	IF arrBetrartHandAktiv[I_nSchutzBer]
		THEN
			stUniAnstgFkt.arrGrdstFkt[0]:= I_arrZuwGrdstFkt[0];
			stUniAnstgFkt.arrGrdstFkt[1]:= I_arrZuwGrdstFkt[1];
			stUniAnstgFkt.arrGrdstFkt[2]:= I_arrZuwGrdstFkt[2];
			stUniAnstgFkt.arrGrdstFkt[3]:= I_arrZuwGrdstFkt[3];
		ELSE
			stUniAnstgFkt.arrGrdstFkt[0]:= 
			stUniAnstgFkt.arrGrdstFkt[1]:=
			stUniAnstgFkt.arrGrdstFkt[2]:=
			stUniAnstgFkt.arrGrdstFkt[3]:= FALSE;
   END_IF
	IF arrBetrartAutomAktiv[I_nSchutzBer] OR TRUE //ToDo
		THEN
			stUniAnstgFkt.arrAutomFkt[0]:= I_arrZuwAutomFkt[0];
			stUniAnstgFkt.arrAutomFkt[1]:= I_arrZuwAutomFkt[1];
			stUniAnstgFkt.arrAutomFkt[2]:= I_arrZuwAutomFkt[2];
			stUniAnstgFkt.arrAutomFkt[3]:= I_arrZuwAutomFkt[3];
		ELSE
			stUniAnstgFkt.arrAutomFkt[0]:= 
			stUniAnstgFkt.arrAutomFkt[1]:= 
			stUniAnstgFkt.arrAutomFkt[2]:= 
			stUniAnstgFkt.arrAutomFkt[3]:= FALSE;
   END_IF

	(**************************************************)	

	stUniAnstgFkt.arrFktAusfg[0]:= stUniAnstgFkt.arrGrdstFkt[0]
										 	 OR stUniAnstgFkt.arrHandFkt[0]
										 	 OR stUniAnstgFkt.arrAutomFkt[0];

	stUniAnstgFkt.arrFktAusfg[1]:= stUniAnstgFkt.arrGrdstFkt[1]
										 	 OR stUniAnstgFkt.arrHandFkt[1]
										 	 OR stUniAnstgFkt.arrAutomFkt[1];

	stUniAnstgFkt.arrFktAusfg[2]:= stUniAnstgFkt.arrGrdstFkt[2]
										 	 OR stUniAnstgFkt.arrHandFkt[2]
										 	 OR stUniAnstgFkt.arrAutomFkt[2];

	stUniAnstgFkt.arrFktAusfg[3]:= stUniAnstgFkt.arrGrdstFkt[3]
										 	 OR stUniAnstgFkt.arrHandFkt[3]
										 	 OR stUniAnstgFkt.arrAutomFkt[3];

	(**************************************************)
END_ACTION

ACTION c_Verstellg:
	(*Antriebstyp "Verstellg." /z.B. FU-Antriebe mit Eil/Schleichbewegung...*)

	(*Verwendete Softkeytasten = 5 (s.Beispiel)*)

   (*       "Handfunktion"       /   "Softkeytaste 1"   /   "Softkeytaste 2"   /   "Softkeytaste 3"   /   "Softkeytaste 4"   /   "Softkeytaste 5"   *)
	(*                                                                          															  								 *) 
	(*----- Verstellantrieb ------/_____zurückfahren_____/_______vorfahren______/_______langsam________/_______schnell________/________Reset_________*)

	(*Softkeyleiste.1		:Funktion ein.-ausschalten Reversierend*)
	(*Softkeyleiste.2		:Funktion ein.-ausschalten             *)
	(*Softkeyleiste.3		:Funktion langsame Drehzahl (SollwMin) *)
	(*Softkeyleiste.4		:Funktion schnelle Drehzahl (SollwVrg) *)
	(*Softkeyleiste.5		:Platzhalter									 *)

	(*Hinweis:
	- Funktion wird durch "VerrHdFkt" gesperrt (z.B. bei Überstandserkennung...)
	- Funktion wird durch "EndlHdFkt/VerzHdFkt" zurückgenommen bzw. umgeschaltet
	*)
	
	(**************************************************)	

	stUniAnstgFkt.bHandAnw0:= IQ_stUniAnstgHMI.stHandFktHMI[1].bySwitch > 0;
	stUniAnstgFkt.bHandAnw1:= IQ_stUniAnstgHMI.stHandFktHMI[2].bySwitch > 0;
	stUniAnstgFkt.bHandAnw2:= IQ_stUniAnstgHMI.stHandFktHMI[3].bySwitch > 0;
	stUniAnstgFkt.bHandAnw3:= IQ_stUniAnstgHMI.stHandFktHMI[4].bySwitch > 0;
	
	IF arrBetrartAutomAktiv[I_nSchutzBer]
		OR I_bResHandFkt
		OR NOT I_bExtReglFrg
		THEN
			stUniAnstgFkt.arrHandFkt[0]:=
			stUniAnstgFkt.arrHandFkt[1]:=
			stUniAnstgFkt.arrHandFkt[2]:=
			stUniAnstgFkt.arrHandFkt[3]:= FALSE;
		ELSE
			IF NOT arrBetrartAutomSpeichn[I_nSchutzBer]
				THEN
					IF NOT arrGrdstlgBetrAktiv[I_nSchutzBer]
						THEN
							 rtrigHandFkt1 (CLK:= stUniAnstgFkt.bHandAnw1);
							 IF rtrigHandFkt1.Q THEN
								 stUniAnstgFkt.arrHandFkt[1]:= NOT stUniAnstgFkt.arrHandFkt[1];
							 END_IF
							 IF NOT arrBetrartHandAktiv[I_nSchutzBer]
								 OR stUniAnstgFkt.arrHandFkt[0]
								 OR I_bVerrHdFktV OR NOT I_bEndlHdFktV THEN
								 stUniAnstgFkt.arrHandFkt[1]:= FALSE;
							 END_IF
	 
							 rtrigHandFkt0 (CLK:= stUniAnstgFkt.bHandAnw0);
							 IF rtrigHandFkt0.Q THEN
								 stUniAnstgFkt.arrHandFkt[0]:= NOT stUniAnstgFkt.arrHandFkt[0];
							 END_IF
							 IF NOT arrBetrartHandAktiv[I_nSchutzBer]
								 OR stUniAnstgFkt.arrHandFkt[1]
								 OR I_bVerrHdFktZ OR NOT I_bEndlHdFktZ THEN
								 stUniAnstgFkt.arrHandFkt[0]:= FALSE;
							 END_IF
	 
							 IF stUniAnstgFkt.bHandAnw3 THEN
								 stUniAnstgFkt.arrHandFkt[3]:= TRUE;
							 END_IF
							 IF NOT arrBetrartHandAktiv[I_nSchutzBer]
								 OR (stUniAnstgFkt.arrHandFkt[1] AND I_bVerzHdFktV)
								 OR (stUniAnstgFkt.arrHandFkt[0] AND I_bVerzHdFktZ)
								 OR stUniAnstgFkt.bHandAnw2 THEN
								 stUniAnstgFkt.arrHandFkt[3]:= FALSE;
							 END_IF
					END_IF
			END_IF
	END_IF

	IF arrBetrartHandAktiv[I_nSchutzBer]
		THEN
			stUniAnstgFkt.nHandStat:= 0;			(*Funktion freigegeben*)
			IF stUniAnstgFkt.arrHandFkt[1]
				THEN
					stUniAnstgFkt.nHandStat:= 2;	(*Handfunktion.2 aktiv*)
			END_IF
			IF stUniAnstgFkt.arrHandFkt[0]
				THEN
					stUniAnstgFkt.nHandStat:= 1;	(*Handfunktion.1 aktiv*)
			END_IF
			IF stUniAnstgFkt.arrHandFkt[3]
				THEN
					stUniAnstgFkt.nHandStat:=
					stUniAnstgFkt.nHandStat + 8;	(*Handfunktion.4 aktiv*)
				ELSE
					stUniAnstgFkt.nHandStat:=
					stUniAnstgFkt.nHandStat + 4;	(*Handfunktion.3 aktiv*)
			END_IF
		ELSE
			stUniAnstgFkt.nHandStat:= 256;		(*Funktion gesperrt*)
	END_IF

	(**************************************************)	

	IF arrBetrartHandAktiv[I_nSchutzBer]
		THEN
			stUniAnstgFkt.arrGrdstFkt[0]:= I_arrZuwGrdstFkt[0];
			stUniAnstgFkt.arrGrdstFkt[1]:= I_arrZuwGrdstFkt[1];
			stUniAnstgFkt.arrGrdstFkt[3]:= I_arrZuwGrdstFkt[2];
		ELSE
			stUniAnstgFkt.arrGrdstFkt[0]:= 
			stUniAnstgFkt.arrGrdstFkt[1]:=
			stUniAnstgFkt.arrGrdstFkt[3]:= FALSE;
   END_IF
	IF arrBetrartAutomAktiv[I_nSchutzBer] OR TRUE //ToDo
		THEN
			stUniAnstgFkt.arrAutomFkt[0]:= I_arrZuwAutomFkt[0];
			stUniAnstgFkt.arrAutomFkt[1]:= I_arrZuwAutomFkt[1];
			stUniAnstgFkt.arrAutomFkt[3]:= I_arrZuwAutomFkt[2];
		ELSE
			stUniAnstgFkt.arrAutomFkt[0]:= 
			stUniAnstgFkt.arrAutomFkt[1]:= 
			stUniAnstgFkt.arrAutomFkt[3]:= FALSE;
   END_IF

	(**************************************************)	

	stUniAnstgFkt.arrFktAusfg[0]:= (stUniAnstgFkt.arrGrdstFkt[0]
										 	 	OR stUniAnstgFkt.arrHandFkt[0]
										 	 	OR stUniAnstgFkt.arrAutomFkt[0])
											AND I_bEndlHdFktZ;

	stUniAnstgFkt.arrFktAusfg[1]:= (stUniAnstgFkt.arrGrdstFkt[1]
										 	 OR stUniAnstgFkt.arrHandFkt[1]
										 	 OR stUniAnstgFkt.arrAutomFkt[1])
											AND I_bEndlHdFktV;

	stUniAnstgFkt.arrFktAusfg[3]:= (stUniAnstgFkt.arrGrdstFkt[3]
												 OR stUniAnstgFkt.arrHandFkt[3]
												 OR stUniAnstgFkt.arrAutomFkt[3])
											AND(( stUniAnstgFkt.arrFktAusfg[0]
													AND NOT I_bVerzHdFktZ)
												OR ( stUniAnstgFkt.arrFktAusfg[1]
													AND NOT I_bVerzHdFktV));

	(**************************************************)
END_ACTION

ACTION d_EilSchleich:
	(*Antriebstyp "EilSchleich" /z.B. FU-Antriebe mit Eil/Schleichachse...*)

	(*Verwendete Softkeytasten = 5 (s.Beispiel)*)

   (*       "Handfunktion"       /   "Softkeytaste 1"   /   "Softkeytaste 2"   /   "Softkeytaste 3"   /   "Softkeytaste 4"   /   "Softkeytaste 5"   *)
	(*                                                                          															  								 *) 
	(*------ Verstellachse -------/____negativ fahren____/____positiv fahren____/_________Frei_________/_________Frei_________/________Reset_________*)
	
	(*Softkeyleiste.1		:Funktion Tastend aktiv /Richtg. Negativ*)
	(*Softkeyleiste.2		:Funktion Tastend aktiv /Richtg. Positiv*)
	(*Softkeyleiste.3		:Platzhalter				 					 *)
	(*Softkeyleiste.4		:Platzhalter				 					 *)
	(*Softkeyleiste.5		:Platzhalter									 *)

	(*Hinweis:
	- Funktion wird durch "VerrHdFkt" gesperrt (z.B. bei Überstandserkennung...)
	*)

	(**************************************************)	

	stUniAnstgFkt.bHandAnw0:= IQ_stUniAnstgHMI.stHandFktHMI[1].bySwitch > 0;
	stUniAnstgFkt.bHandAnw1:= IQ_stUniAnstgHMI.stHandFktHMI[2].bySwitch > 0;
	
	IF arrBetrartAutomAktiv[I_nSchutzBer]
		OR NOT I_bExtReglFrg
		THEN
			stUniAnstgFkt.arrHandFkt[0]:=
			stUniAnstgFkt.arrHandFkt[1]:= FALSE;
		ELSE
			IF NOT arrBetrartAutomSpeichn[I_nSchutzBer] THEN
				IF NOT arrGrdstlgBetrAktiv[I_nSchutzBer] THEN
					stUniAnstgFkt.arrHandFkt[1]:= arrBetrartHandAktiv[I_nSchutzBer]
													  		AND stUniAnstgFkt.bHandAnw1
													  		AND NOT stUniAnstgFkt.bHandAnw0
													  		AND NOT I_bVerrHdFktV	
													  		AND I_RefAchse.stFreigb.bVorsFrgPos;
					stUniAnstgFkt.arrHandFkt[0]:= arrBetrartHandAktiv[I_nSchutzBer]
													  		AND stUniAnstgFkt.bHandAnw0
													  		AND NOT stUniAnstgFkt.bHandAnw1
													  		AND NOT I_bVerrHdFktZ
													  		AND I_RefAchse.stFreigb.bVorsFrgNeg;
				END_IF
			END_IF
	END_IF

	IF arrBetrartHandAktiv[I_nSchutzBer]
		THEN
			stUniAnstgFkt.nHandStat:= 0;			(*Funktion freigegeben*)
			IF stUniAnstgFkt.arrHandFkt[1]
				THEN
					stUniAnstgFkt.nHandStat:= 2;	(*Handfunktion.2 aktiv*)
			END_IF
			IF stUniAnstgFkt.arrHandFkt[0]
				THEN
					stUniAnstgFkt.nHandStat:= 1;	(*Handfunktion.1 aktiv*)
			END_IF
		ELSE
			stUniAnstgFkt.nHandStat:= 256;		(*Funktion gesperrt*)
	END_IF

	(**************************************************)	
	
	I_RefAchse.stStatus.bAchseBTB	:= Q_bAbfrStatUmr;

	I_RefAchse.stGrdfkt.bHdfkt_pos:=	stUniAnstgFkt.arrHandFkt[1];
	I_RefAchse.stGrdfkt.bHdfkt_neg:=	stUniAnstgFkt.arrHandFkt[0];

	(**************************************************)
END_ACTION

ACTION u_AggEinlZykl:
	(*Inbetriebnahme HF-Aggregate (Einlaufphasen für optimale Fettverteilung)*)

IF NOT I_bAnwEinlZykl
THEN
	nStepEinlZykl	:= 0;		 

	RETURN;
END_IF

	(**************************************************)	

CASE nStepEinlZykl OF
	
0:
	
	tonEinlZyklPhase (IN:= FALSE);
	nEinlZyklPhase:= 1;

	IF stUniAnstgFkt.arrHandFkt[1]
	THEN	// Antrieb muss in den Handfunktionen eingeschaltet werden, damit der Erste Warmlaufzyklus durchgeführt wird.
		nStepEinlZykl:= 100;
   END_IF

100, 110, 120, 130, 140, 150, 160, 170, 180, 190, 200, 210, 220, 230, 240, 250, 260, 270, 280, 290:
	//Einlaufphasen 1-20:

	Q_bRichtVrgV	:= arrEinlZyklDrehz[nEinlZyklPhase].0;
	Q_bSollwVrg_N11:= arrEinlZyklDrehz[nEinlZyklPhase].1;
	Q_bSollwVrg_N12:= arrEinlZyklDrehz[nEinlZyklPhase].2;

	tonEinlZyklPhase (IN:= stUniAnstgFkt.arrHandFkt[1],
							PT:= arrEinlZyklPhase[nEinlZyklPhase]);

	IF tonEinlZyklPhase.Q
	THEN
		tonEinlZyklPhase (IN:= FALSE);
		nEinlZyklPhase:= nEinlZyklPhase + 1;
		
		nStepEinlZykl:= nStepEinlZykl + 10;		 
	END_IF	

	IF NOT stUniAnstgFkt.arrHandFkt[1]
	THEN
		nStepEinlZykl:= 0;		 
   END_IF
	
300:
	//Ende Einlaufzyklus
	nStepEinlZykl:= nStepEinlZykl;		 
	
END_CASE

	
	(**************************************************)
END_ACTION

ACTION v_AggBetrZykl:
	(*Betriebszyklen HF-Aggregate (Warmlaufphasen z. Verschleißminderung)*)

	IF I_bAnwEinlZykl THEN
		nStepBetrZykl	:= 0;		 
		bHochlZyklStart:=
		bHochlZyklEnde	:= FALSE;

		RETURN;
	END_IF

	(**************************************************)	

	IF stUniAnstgFkt.arrFktAusfg[1]	//Optional weitere Bedingungen? 
		OR I_bStandbyBetr
	THEN //Betriebszyklus start
		bHochlZyklStart	:= TRUE;	

	ELSIF FALSE (*Optional*)
	THEN //Betriebszyklus stop
		bHochlZyklStart	:= FALSE;	

		nStepBetrZykl	:= 0;		 

	ELSIF NOT stUniAnstgFkt.arrFktAusfg[1]
		AND NOT I_bStandbyBetr
	THEN //Betriebszyklus halt 
		bHochlZyklStart	:= FALSE;	

	END_IF

	(**************************************************)	
	
	CASE nStepBetrZykl OF
0:
	//Initialisierung:
	nDrehzBetrZykl:= 0;

	bHochlZyklEnde:= FALSE;	
	
	tonBetrZyklPhase (IN:= FALSE);
	nBetrZyklPhase:= 0;
	
	IF bHochlZyklStart THEN
		nStepBetrZykl:= 100;		 
   END_IF

100, 200, 300:
	//Hochlaufphasen 1-3:
	nBetrZyklPhase:= nStepBetrZykl / 100; 

	Q_bRichtVrgV	:= nBetrZyklPhase = 1;
	Q_bSollwVrg_N11:= nBetrZyklPhase = 2;
	Q_bSollwVrg_N12:= nBetrZyklPhase = 3;
	
	tonBetrZyklPhase (IN:= bHochlZyklStart,
							PT:= I_arrBetrZyklPhase[nBetrZyklPhase]);
	
	IF tonBetrZyklPhase.Q THEN
		tonBetrZyklPhase (IN:= FALSE);
		
		nStepBetrZykl:= nStepBetrZykl + 100;		 

	ELSIF NOT bHochlZyklStart THEN
		tonBetrZyklPhase (IN:= FALSE);
		
		nStepBetrZykl:= nStepBetrZykl * -1;		 
	END_IF	

400:
	//Ende Hochlaufzyklus => Betriebsbereit
	nBetrZyklPhase:= nStepBetrZykl / 100; 

	bHochlZyklEnde:= TRUE;	
	
	IF stUniAnstgFkt.arrFktAusfg[1]
	THEN	//Bearbeitungsdrehzahl
		Q_bRichtVrgV	:= TRUE;
		Q_bSollwVrg_N11:= FALSE;
		Q_bSollwVrg_N12:= TRUE;
	ELSE	//Leerlaufdrehzahl
		Q_bRichtVrgV	:= TRUE;
		Q_bSollwVrg_N11:= FALSE;
		Q_bSollwVrg_N12:= FALSE;
   END_IF

	tonBetrZyklPhase (IN:= NOT bHochlZyklStart,
							PT:= I_arrBetrZyklPhase[nBetrZyklPhase]);
	
	IF tonBetrZyklPhase.Q THEN
		tonBetrZyklPhase (IN:= FALSE);

		bHochlZyklEnde:= FALSE;	
		
		nStepBetrZykl:= 500;		 
	END_IF

500:
	//Stillstandphase > 15min
	tonBetrZyklPhase (IN:= TRUE,
							PT:= I_tPause);
	
	IF tonBetrZyklPhase.Q THEN
		tonBetrZyklPhase (IN:= FALSE);
	
		nStepBetrZykl:= 0;		 

	ELSIF bHochlZyklStart THEN 
		tonBetrZyklPhase (IN:= FALSE);

		IF tonBetrZyklPhase.ET > (I_tPause/2) //Halbe Stillstandszeit
			THEN		
				nStepBetrZykl:= 300; //Erneuter Hochlauf ab Phase 3 			 
			ELSE
				nStepBetrZykl:= 400; //Direkt wieder Betriebsbereit		 
	  END_IF
	END_IF	
	
	nDrehzBetrZykl:= 0;

ELSE
	//Hochlaufphase Unterbrochen 
	tonBetrZyklPhase (IN:= TRUE,
							PT:= T#15S);
	
	IF tonBetrZyklPhase.Q THEN
		tonBetrZyklPhase (IN:= FALSE);

		CASE nStepBetrZykl OF
		-100:	nStepBetrZykl:= 0;	
		-200:	nStepBetrZykl:= 100;	
		-300:	nStepBetrZykl:= 200;	
	  	END_CASE

	ELSIF bHochlZyklStart THEN 
		tonBetrZyklPhase (IN:= FALSE);

		nStepBetrZykl:= nStepBetrZykl * -1;		 

	END_IF	

END_CASE
	
	(**************************************************)
END_ACTION

ACTION w_InOutSEW:

	(**************************************************)	
	(*EtherCAT-Anschaltung*)	

	bUmrStat	:= I_bUmrStat;

	IF I_eAntriebTyp = E_AntriebTyp.eAggregat
	THEN
		IF stUniAnstgFkt.arrFktAusfg[1] 
		THEN
			Q_bRichtVrgV	:= TRUE;
		ELSE
			Q_bRichtVrgV	:= FALSE;
		END_IF
		
	ELSIF I_eAntriebTyp = E_AntriebTyp.eTransport
		OR I_eAntriebTyp = E_AntriebTyp.eVerstellg
	THEN
	
		Q_bSollwVrg_N11		:= stUniAnstgFkt.arrFktAusfg[2];
		Q_bSollwVrg_N12		:= stUniAnstgFkt.arrFktAusfg[3];
		
		IF stUniAnstgFkt.arrFktAusfg[0]
		THEN
			Q_bRichtVrgR	:= TRUE;
			Q_bRichtVrgV	:= FALSE;
		ELSIF stUniAnstgFkt.arrFktAusfg[1]
		THEN
			Q_bRichtVrgV	:= TRUE;
			Q_bRichtVrgR	:= FALSE;
		ELSE
			Q_bRichtVrgV	:= FALSE;
			Q_bRichtVrgR	:= FALSE;
			Q_bSollwVrg_N11:= FALSE;
			Q_bSollwVrg_N12:= FALSE;
		END_IF
		
	ELSIF I_eAntriebTyp = E_AntriebTyp.eEilSchleich
	THEN
		Q_bRichtVrgV	:= I_RefAxis.Status.PositiveDirection
								AND I_RefAxis.NcToPlc.SetVelo > 0;
		Q_bRichtVrgR	:= I_RefAxis.Status.NegativeDirection
								AND I_RefAxis.NcToPlc.SetVelo > 0;
		Q_bSollwVrg_N11		:= I_RefAxis.NcToPlc.SetVelo > 50
								AND I_RefAchse.stStatus.bInReferz;
		
	ELSIF I_eAntriebTyp = E_AntriebTyp.eAggregatHF
	THEN
		IF stUniAnstgFkt.arrFktAusfg[1]
		THEN
			Q_bRichtVrgV	:= TRUE;
		ELSE
			Q_bRichtVrgV	:= FALSE;
		END_IF
   END_IF

	IF NOT arrAntrGruppeFrg[I_nSchutzBer] (*Allg. Freigabe /..Fräser Abbremsen*)
	THEN
		Q_bRichtVrgR	:= FALSE;
		Q_bRichtVrgV	:= FALSE;
		Q_bSollwVrg_N11:= FALSE;	
		Q_bSollwVrg_N12:= FALSE;		 
	END_IF

	(**)

	Q_bAbfrStatUmr		:= bUmrStat;

// ENDE
END_ACTION

ACTION x_AusgZuw:
	
	(**************************************************)	
	(*Ausgänge zuweisen*)
										
	CASE I_nAntrEinsGrp OF
1:	Q_bAnstNetzUmr:= arrAntrGruppe1Ein[I_nSchutzBer]
					  	  AND bVersEingAusgSchaltsOk;

2:	Q_bAnstNetzUmr:= arrAntrGruppe2Ein[I_nSchutzBer]
					  	  AND bVersEingAusgSchaltsOk;

3:	Q_bAnstNetzUmr:= arrAntrGruppe3Ein[I_nSchutzBer]
					  	  AND bVersEingAusgSchaltsOk;
	END_CASE

	Q_bAnstReglFrg:= arrAntrGruppeFrg[I_nSchutzBer]
						  AND I_bExtReglFrg
					  	  AND bUmrStat
					  	  AND bVersEingAusgSchaltsOk;

	(**************************************************)	
;
END_ACTION

ACTION y_ZustAnzg:
	
	(**************************************************)	
	(*Zustände anzeigen*)

	CASE I_eAntriebTyp OF

E_AntriebTyp.eAggregat:	// nur zwei Handfunktionen aktiv

	IF stUniAnstgFkt.nHandStat = 1	(*Handfunktion.1 aktiv*)
	THEN
		IQ_stUniAnstgHMI.stHandFktHMI[1].sColour:= cGruenAsString;
		IQ_stUniAnstgHMI.stHandFktHMI[2].sColour:= cDefaultAsString;
		IQ_stUniAnstgHMI.stHandFktHMI[1].sText:= 'ausgeschaltet';
		IQ_stUniAnstgHMI.stHandFktHMI[2].sText:= 'einschalten';
   END_IF
	
	IF stUniAnstgFkt.nHandStat = 2	(*Handfunktion.2 aktiv*)
	THEN
		IQ_stUniAnstgHMI.stHandFktHMI[1].sColour:= cDefaultAsString;
		IQ_stUniAnstgHMI.stHandFktHMI[2].sColour:= cGruenAsString;
		IQ_stUniAnstgHMI.stHandFktHMI[1].sText:= 'ausschalten';
		IQ_stUniAnstgHMI.stHandFktHMI[2].sText:= 'eingeschaltet';
   END_IF
	
	IQ_stUniAnstgHMI.stHandFktHMI[3].sColour:= cDefaultAsString;
	IQ_stUniAnstgHMI.stHandFktHMI[3].sText:= ' ';
	IQ_stUniAnstgHMI.stHandFktHMI[4].sColour:= cDefaultAsString;
	IQ_stUniAnstgHMI.stHandFktHMI[4].sText:= ' ';
	IQ_stUniAnstgHMI.stHandFktHMI[5].sColour:= cDefaultAsString;
	IQ_stUniAnstgHMI.stHandFktHMI[5].sText:= ' ';

	IF stUniAnstgFkt.nHandStat = 256	(*Funktion gesperrt*)
	THEN
		IQ_stUniAnstgHMI.stHandFktHMI[1].sText:= 'ausgeschaltet';
		IQ_stUniAnstgHMI.stHandFktHMI[2].sText:= 'einschalten';
		IQ_stUniAnstgHMI.stHandFktHMI[1].sColour:= cDefaultAsString;
		IQ_stUniAnstgHMI.stHandFktHMI[2].sColour:= cDefaultAsString;
		IQ_stUniAnstgHMI.stHandFktHMI[1].sColour:=
		IQ_stUniAnstgHMI.stHandFktHMI[2].sColour:=cDefaultAsString;
		IQ_stUniAnstgHMI.stHandFktHMI[1].byStatus:=
		IQ_stUniAnstgHMI.stHandFktHMI[2].byStatus:=
		IQ_stUniAnstgHMI.stHandFktHMI[3].byStatus:=
		IQ_stUniAnstgHMI.stHandFktHMI[4].byStatus:=
		IQ_stUniAnstgHMI.stHandFktHMI[5].byStatus:= 1;
	ELSE
		IQ_stUniAnstgHMI.stHandFktHMI[1].byStatus:=
		IQ_stUniAnstgHMI.stHandFktHMI[2].byStatus:= 0;
		IQ_stUniAnstgHMI.stHandFktHMI[3].byStatus:=	// Ist immer deaktiviert
		IQ_stUniAnstgHMI.stHandFktHMI[4].byStatus:=	// Ist immer deaktiviert
		IQ_stUniAnstgHMI.stHandFktHMI[5].byStatus:= 1;	// Ist immer deaktiviert
   END_IF

E_AntriebTyp.eAggregatHF:

	IF stUniAnstgFkt.nHandStat = 1	(*Handfunktion.1 aktiv*)
	THEN
		IQ_stUniAnstgHMI.stHandFktHMI[1].sColour:= cGruenAsString; //eventl.: cRot;
		IQ_stUniAnstgHMI.stHandFktHMI[2].sColour:= cDefaultAsString;
		IQ_stUniAnstgHMI.stHandFktHMI[1].sText:= 'ausgeschaltet';
		IQ_stUniAnstgHMI.stHandFktHMI[2].sText:= 'einschalten';
   END_IF
	
	IF stUniAnstgFkt.nHandStat = 2	(*Handfunktion.2 aktiv*)
	THEN
		IQ_stUniAnstgHMI.stHandFktHMI[1].sColour:= cDefaultAsString;
		IQ_stUniAnstgHMI.stHandFktHMI[2].sColour:= cGruenAsString;
		IQ_stUniAnstgHMI.stHandFktHMI[1].sText:= 'ausschalten';
		IQ_stUniAnstgHMI.stHandFktHMI[2].sText:= 'eingeschaltet';
   END_IF
	
	IQ_stUniAnstgHMI.stHandFktHMI[3].sColour:= cDefaultAsString;
	IQ_stUniAnstgHMI.stHandFktHMI[3].sText:= 'Sollwert 1';
	IQ_stUniAnstgHMI.stHandFktHMI[4].sColour:= cDefaultAsString;
	IQ_stUniAnstgHMI.stHandFktHMI[4].sText:= 'Sollwert 2';
	IQ_stUniAnstgHMI.stHandFktHMI[5].sColour:= cDefaultAsString;
	IQ_stUniAnstgHMI.stHandFktHMI[5].sText:= 'Sollwert 3';

	IF stUniAnstgFkt.nHandStat = 256	(*Funktion gesperrt*)
	THEN
		IQ_stUniAnstgHMI.stHandFktHMI[1].sText:= 'ausgeschaltet';
		IQ_stUniAnstgHMI.stHandFktHMI[2].sText:= 'einschalten';
		IQ_stUniAnstgHMI.stHandFktHMI[1].sColour:= cDefaultAsString;
		IQ_stUniAnstgHMI.stHandFktHMI[2].sColour:= cDefaultAsString;
		IQ_stUniAnstgHMI.stHandFktHMI[1].sColour:=
		IQ_stUniAnstgHMI.stHandFktHMI[2].sColour:= cDefaultAsString;
		IQ_stUniAnstgHMI.stHandFktHMI[1].byStatus:=
		IQ_stUniAnstgHMI.stHandFktHMI[2].byStatus:=
		IQ_stUniAnstgHMI.stHandFktHMI[3].byStatus:=
		IQ_stUniAnstgHMI.stHandFktHMI[4].byStatus:=
		IQ_stUniAnstgHMI.stHandFktHMI[5].byStatus:= 1;
	ELSE
		IQ_stUniAnstgHMI.stHandFktHMI[1].byStatus:=
		IQ_stUniAnstgHMI.stHandFktHMI[2].byStatus:=
		IQ_stUniAnstgHMI.stHandFktHMI[3].byStatus:=
		IQ_stUniAnstgHMI.stHandFktHMI[4].byStatus:=
		IQ_stUniAnstgHMI.stHandFktHMI[5].byStatus:= 0;
   END_IF

E_AntriebTyp.eTransport:

	IF stUniAnstgFkt.arrHandFkt[0] (*Handfunktion.1 aktiv*)
	THEN
		IQ_stUniAnstgHMI.stHandFktHMI[1].sColour:= cGruenAsString;
		IQ_stUniAnstgHMI.stHandFktHMI[1].sText:= 'ausschalten';
	ELSE
		IQ_stUniAnstgHMI.stHandFktHMI[1].sColour:= cDefaultAsString;
		IQ_stUniAnstgHMI.stHandFktHMI[1].sText:= 'zurück';
		
		IF stUniAnstgFkt.arrHandFkt[1]
		THEN
			IQ_stUniAnstgHMI.stHandFktHMI[1].sText:= ' ';
		END_IF
   END_IF
	
	IF stUniAnstgFkt.arrHandFkt[1]	(*Handfunktion.2 aktiv*)
	THEN		 
		IQ_stUniAnstgHMI.stHandFktHMI[2].sColour:= cGruenAsString;
		IQ_stUniAnstgHMI.stHandFktHMI[2].sText:= 'ausschalten';
	ELSE
		IQ_stUniAnstgHMI.stHandFktHMI[2].sColour:= cDefaultAsString;
		IQ_stUniAnstgHMI.stHandFktHMI[2].sText:= 'vor';
		
		IF stUniAnstgFkt.arrHandFkt[0]
		THEN	// Zurückfahren ist angewählt
			IQ_stUniAnstgHMI.stHandFktHMI[2].sText:= ' ';
		END_IF
   END_IF
	
	// Handfunktion 3
	IF stUniAnstgFkt.arrHandFkt[2]	// nur Handfunktion.3 aktiv, nicht 4
		AND NOT stUniAnstgFkt.arrHandFkt[3]
	THEN
		IQ_stUniAnstgHMI.stHandFktHMI[3].sColour:= cGruenAsString;
		IQ_stUniAnstgHMI.stHandFktHMI[3].sText:= 'V = N11';
		
	ELSIF stUniAnstgFkt.arrHandFkt[2]	// nur Handfunktion.3 und 4 aktiv
		AND stUniAnstgFkt.arrHandFkt[3]
	THEN
		IQ_stUniAnstgHMI.stHandFktHMI[3].sColour:= cGruenAsString;
		IQ_stUniAnstgHMI.stHandFktHMI[3].sText:= 'V = N13';
		
	ELSIF NOT stUniAnstgFkt.arrHandFkt[2]	// nur Handfunktion.4 und nicht 3 aktiv
		AND stUniAnstgFkt.arrHandFkt[3]
	THEN
		IQ_stUniAnstgHMI.stHandFktHMI[3].sColour:= cDefaultAsString;
		IQ_stUniAnstgHMI.stHandFktHMI[3].sText:= 'V = N12';
	ELSE
		IQ_stUniAnstgHMI.stHandFktHMI[3].sColour:= cDefaultAsString;
		IQ_stUniAnstgHMI.stHandFktHMI[3].sText:= 'V = min';
   END_IF
	
	// Handfunktion 4
	IF NOT stUniAnstgFkt.arrHandFkt[2]	(* nur Handfunktion.4 aktiv, nicht 3*)
		AND stUniAnstgFkt.arrHandFkt[3]
	THEN
		IQ_stUniAnstgHMI.stHandFktHMI[4].sColour:= cGruenAsString;
		IQ_stUniAnstgHMI.stHandFktHMI[4].sText:= 'V = N12';
		
	ELSIF stUniAnstgFkt.arrHandFkt[2]	// nur Handfunktion.3 und 4 aktiv
		AND stUniAnstgFkt.arrHandFkt[3]
	THEN
		IQ_stUniAnstgHMI.stHandFktHMI[4].sColour:= cGruenAsString;
		IQ_stUniAnstgHMI.stHandFktHMI[4].sText:= 'V = N13';
		
	ELSIF stUniAnstgFkt.arrHandFkt[2]	// nur Handfunktion 3 und nicht 4 aktiv
		AND NOT stUniAnstgFkt.arrHandFkt[3]
	THEN
		IQ_stUniAnstgHMI.stHandFktHMI[4].sColour:= cDefaultAsString;
		IQ_stUniAnstgHMI.stHandFktHMI[4].sText:= 'V = N11';
	ELSE
		IQ_stUniAnstgHMI.stHandFktHMI[4].sColour:= cDefaultAsString;
		IQ_stUniAnstgHMI.stHandFktHMI[4].sText:= 'V = min';
   END_IF

	IF stUniAnstgFkt.nHandStat = 256	(*Funktion gesperrt*)
	THEN
		IQ_stUniAnstgHMI.stHandFktHMI[1].sText:= 'zurück';
		IQ_stUniAnstgHMI.stHandFktHMI[2].sText:= 'vor';
		IQ_stUniAnstgHMI.stHandFktHMI[1].byStatus:=
		IQ_stUniAnstgHMI.stHandFktHMI[2].byStatus:=
		IQ_stUniAnstgHMI.stHandFktHMI[3].byStatus:=
		IQ_stUniAnstgHMI.stHandFktHMI[4].byStatus:=
		IQ_stUniAnstgHMI.stHandFktHMI[5].byStatus:= 1;
	ELSE
		IQ_stUniAnstgHMI.stHandFktHMI[1].byStatus:=
		IQ_stUniAnstgHMI.stHandFktHMI[2].byStatus:=
		IQ_stUniAnstgHMI.stHandFktHMI[3].byStatus:=
		IQ_stUniAnstgHMI.stHandFktHMI[4].byStatus:= 0;
		IQ_stUniAnstgHMI.stHandFktHMI[5].byStatus:= 1;	// Ist immer deaktiviert
   END_IF

E_AntriebTyp.eVerstellg:
	
	IF GETBIT32 (TO_DWORD(stUniAnstgFkt.nHandStat), 0)	(*Handfunktion.1 aktiv*)
	THEN
		IQ_stUniAnstgHMI.stHandFktHMI[1].sColour:= cGruenAsString;
		IQ_stUniAnstgHMI.stHandFktHMI[1].sText:= 'zurückfahren';
	ELSE
		IQ_stUniAnstgHMI.stHandFktHMI[1].sColour:= cDefaultAsString;
		
		IF NOT I_bEndlHdFktZ 
		THEN
			IQ_stUniAnstgHMI.stHandFktHMI[1].sColour:= cGruenAsString;
			IQ_stUniAnstgHMI.stHandFktHMI[1].sText:= 'zurückgefahren';
		ELSE
			IQ_stUniAnstgHMI.stHandFktHMI[1].sColour:= cDefaultAsString;
			IQ_stUniAnstgHMI.stHandFktHMI[1].sText:= 'zurückfahren';
		END_IF
   END_IF
	
	IF GETBIT32 (TO_DWORD(stUniAnstgFkt.nHandStat), 1)	(*Handfunktion.2 aktiv*)
	THEN		 
		IQ_stUniAnstgHMI.stHandFktHMI[2].sColour:= cGruenAsString;
		IQ_stUniAnstgHMI.stHandFktHMI[2].sText:= 'vorfahren';
	ELSE
		IF NOT I_bEndlHdFktV 
		THEN
			IQ_stUniAnstgHMI.stHandFktHMI[2].sColour:= cGruenAsString;
			IQ_stUniAnstgHMI.stHandFktHMI[2].sText:= 'vorgefahren';
		ELSE
			IQ_stUniAnstgHMI.stHandFktHMI[2].sColour:= cDefaultAsString;
			IQ_stUniAnstgHMI.stHandFktHMI[2].sText:= 'vorfahren';
		END_IF
   END_IF
	
	IF GETBIT32 (TO_DWORD(stUniAnstgFkt.nHandStat), 2)	(*Handfunktion.3 aktiv*)
	THEN
		IQ_stUniAnstgHMI.stHandFktHMI[3].sColour:= cGruenAsString;
		IQ_stUniAnstgHMI.stHandFktHMI[3].sText:= 'langsam';
	ELSE
		IQ_stUniAnstgHMI.stHandFktHMI[3].sColour:= cDefaultAsString;
		IQ_stUniAnstgHMI.stHandFktHMI[3].sText:= 'langsam';
   END_IF
	
	IF GETBIT32 (TO_DWORD(stUniAnstgFkt.nHandStat), 3)	(*Handfunktion.4 aktiv*)
	THEN
		IQ_stUniAnstgHMI.stHandFktHMI[4].sColour:= cGruenAsString;
		IQ_stUniAnstgHMI.stHandFktHMI[4].sText:= 'schnell';
	ELSE
		IQ_stUniAnstgHMI.stHandFktHMI[4].sColour:= cDefaultAsString;
		IQ_stUniAnstgHMI.stHandFktHMI[4].sText:= 'schnell';
   END_IF

	IF stUniAnstgFkt.nHandStat = 256	(*Funktion gesperrt*)
	THEN
		IF NOT I_bEndlHdFktZ 
		THEN
			IQ_stUniAnstgHMI.stHandFktHMI[1].sColour:= cGruenAsString;
			IQ_stUniAnstgHMI.stHandFktHMI[1].sText:= 'zurückgefahren';
		ELSE
			IQ_stUniAnstgHMI.stHandFktHMI[1].sColour:= cDefaultAsString;
			IQ_stUniAnstgHMI.stHandFktHMI[1].sText:= 'zurückfahren';
		END_IF
		IF NOT I_bEndlHdFktV 
		THEN
			IQ_stUniAnstgHMI.stHandFktHMI[2].sColour:= cGruenAsString;
			IQ_stUniAnstgHMI.stHandFktHMI[2].sText:= 'vorgefahren';
		ELSE
			IQ_stUniAnstgHMI.stHandFktHMI[2].sColour:= cDefaultAsString;
			IQ_stUniAnstgHMI.stHandFktHMI[2].sText:= 'vorfahren';
		END_IF
		IQ_stUniAnstgHMI.stHandFktHMI[3].sText:= 'langsam';
		IQ_stUniAnstgHMI.stHandFktHMI[4].sText:= 'schnell';
		IQ_stUniAnstgHMI.stHandFktHMI[1].byStatus:=
		IQ_stUniAnstgHMI.stHandFktHMI[2].byStatus:=
		IQ_stUniAnstgHMI.stHandFktHMI[3].byStatus:=
		IQ_stUniAnstgHMI.stHandFktHMI[4].byStatus:=
		IQ_stUniAnstgHMI.stHandFktHMI[5].byStatus:= 1;
	ELSE
		IQ_stUniAnstgHMI.stHandFktHMI[1].byStatus:=
		IQ_stUniAnstgHMI.stHandFktHMI[2].byStatus:=
		IQ_stUniAnstgHMI.stHandFktHMI[3].byStatus:=
		IQ_stUniAnstgHMI.stHandFktHMI[4].byStatus:= 0;
		IQ_stUniAnstgHMI.stHandFktHMI[5].byStatus:= 1;	// Ist immer deaktiviert
   END_IF

E_AntriebTyp.eEilSchleich:
	
	IF stUniAnstgFkt.nHandStat = 1	(*Handfunktion.1 aktiv*)
	THEN
		IQ_stUniAnstgHMI.stHandFktHMI[1].sColour:= cGruenAsString;
		IQ_stUniAnstgHMI.stHandFktHMI[1].sText:= 'negativ fahren';
	ELSE
		IQ_stUniAnstgHMI.stHandFktHMI[1].sColour:= cDefaultAsString;
		IQ_stUniAnstgHMI.stHandFktHMI[1].sText:= 'negativ fahren';
   END_IF
	
	IF stUniAnstgFkt.nHandStat = 2	(*Handfunktion.2 aktiv*)
	THEN		 
		IQ_stUniAnstgHMI.stHandFktHMI[2].sColour:= cGruenAsString;
		IQ_stUniAnstgHMI.stHandFktHMI[2].sText:= 'positiv fahren';
	ELSE
		IQ_stUniAnstgHMI.stHandFktHMI[2].sColour:= cDefaultAsString;
		IQ_stUniAnstgHMI.stHandFktHMI[2].sText:= 'positiv fahren';
   END_IF
	
	IQ_stUniAnstgHMI.stHandFktHMI[3].sColour:= cDefaultAsString;
	IQ_stUniAnstgHMI.stHandFktHMI[3].sText:= ' ';
	IQ_stUniAnstgHMI.stHandFktHMI[4].sColour:= cDefaultAsString;
	IQ_stUniAnstgHMI.stHandFktHMI[4].sText:= ' ';
	IQ_stUniAnstgHMI.stHandFktHMI[5].sColour:= cDefaultAsString;
	IQ_stUniAnstgHMI.stHandFktHMI[5].sText:= ' ';

	IF stUniAnstgFkt.nHandStat = 256	(*Funktion gesperrt*)
	THEN
		IQ_stUniAnstgHMI.stHandFktHMI[1].sText:= 'negativ fahren';
		IQ_stUniAnstgHMI.stHandFktHMI[2].sText:= 'positiv fahren';
		IQ_stUniAnstgHMI.stHandFktHMI[1].sColour:=
		IQ_stUniAnstgHMI.stHandFktHMI[2].sColour:=cDefaultAsString;
		IQ_stUniAnstgHMI.stHandFktHMI[1].byStatus:=
		IQ_stUniAnstgHMI.stHandFktHMI[2].byStatus:=
		IQ_stUniAnstgHMI.stHandFktHMI[3].byStatus:=
		IQ_stUniAnstgHMI.stHandFktHMI[4].byStatus:=
		IQ_stUniAnstgHMI.stHandFktHMI[5].byStatus:= 1;
	ELSE
		IQ_stUniAnstgHMI.stHandFktHMI[1].byStatus:=
		IQ_stUniAnstgHMI.stHandFktHMI[2].byStatus:= 0;
		IQ_stUniAnstgHMI.stHandFktHMI[3].byStatus:=
		IQ_stUniAnstgHMI.stHandFktHMI[4].byStatus:=
		IQ_stUniAnstgHMI.stHandFktHMI[5].byStatus:= 1;
   END_IF
	
   END_CASE

	(**************************************************)
END_ACTION

ACTION z_FehlMeld:

	(**************************************************)	
	(*Meldungen ausgeben*)

	IQ_stUniAnstgHMI.stMeldAusgHMI.SourceID			:= 0;	// Nicht mehr verwendet
	IQ_stUniAnstgHMI.stMeldAusgHMI.SourceName			:= I_sStatName;
	IQ_stUniAnstgHMI.stMeldAusgHMI.sAktorName			:= I_sAktorName;
	
	IF I_sAktorBMK <> ''
	THEN	// I_sAktorBMK ist beschrieben. Damit wird der String als BMK genommen
		IQ_stUniAnstgHMI.stMeldAusgHMI.sBMK	:= I_sAktorBMK;
	ELSE	// Der Kommentar von VARINFO wird als BMK genommen
		IQ_stUniAnstgHMI.stMeldAusgHMI.sBMK	:= I_stVarInfoBMK.Comment;
	END_IF

	IQ_stUniAnstgHMI.stMeldAusgHMI.bMeldNichtBtb		:= (arrAntrGruppeFrg[I_nSchutzBer]
					  	  													AND NOT bUmrStat
					  	  													AND bVersEingAusgSchaltsOk)
																		OR bTestMeldAntr;

	IF I_eAntriebTyp = eEilSchleich
	THEN
		IQ_stUniAnstgHMI.stMeldAusgHMI.bMeldNichtReferenz		:= (NOT I_RefAchse.stStatus.bInReferz
																					AND NOT I_RefAchse.stGrdfkt.bRefrz_ausf)
																					OR bTestMeldAntrEilSchleich;
		IQ_stUniAnstgHMI.stMeldAusgHMI.bMeldReffahrtStart		:= I_RefAchse.stGrdfkt.bRefrz_ausf
																					OR bTestMeldAntrEilSchleich;
	END_IF

	IF I_eAntriebTyp = eVerstellg
	THEN
		tonMeldLaufzeit0(	IN := stUniAnstgFkt.arrHandFkt[0]
										AND NOT I_bEndlHdFktZ,
								PT := I_tLaufzeitMeld);
		tonMeldLaufzeit1(	IN := stUniAnstgFkt.arrHandFkt[1]
										AND NOT I_bEndlHdFktV,
								PT := I_tLaufzeitMeld);
		IQ_stUniAnstgHMI.stMeldAusgHMI.bMeldLaufzeit0		:= tonMeldLaufzeit0.Q
																					OR bTestMeldAntrVerstellg;
		IQ_stUniAnstgHMI.stMeldAusgHMI.bMeldLaufzeit1		:= tonMeldLaufzeit1.Q
																					OR bTestMeldAntrVerstellg;
	END_IF
	
	
	(*Zus. Hinweise HF-Aggregate*)
	IF bTestMeldAntrHF
	THEN
		IQ_stUniAnstgHMI.stMeldAusgHMI.bMeldEinlZyklAktiv	:=
		IQ_stUniAnstgHMI.stMeldAusgHMI.bMeldEinlZyklBeendet:=
		IQ_stUniAnstgHMI.stMeldAusgHMI.bMeldWarmlaufZykl	:= TRUE;
	ELSIF nStepEinlZykl > 1 AND nStepEinlZykl < 300 
	THEN 						
		IQ_stUniAnstgHMI.stMeldAusgHMI.bMeldEinlZyklAktiv	:= TRUE;
		IQ_stUniAnstgHMI.stMeldAusgHMI.bMeldEinlZyklBeendet:=
		IQ_stUniAnstgHMI.stMeldAusgHMI.bMeldWarmlaufZykl	:= FALSE;
	ELSIF nStepEinlZykl = 300 
	THEN
		IQ_stUniAnstgHMI.stMeldAusgHMI.bMeldEinlZyklAktiv	:= FALSE;
		IQ_stUniAnstgHMI.stMeldAusgHMI.bMeldEinlZyklBeendet:= TRUE;
		IQ_stUniAnstgHMI.stMeldAusgHMI.bMeldWarmlaufZykl	:= FALSE;
	ELSIF (nStepBetrZykl > 1 AND nStepBetrZykl < 400)
      OR (nStepBetrZykl < 0) 
	THEN
		IQ_stUniAnstgHMI.stMeldAusgHMI.bMeldEinlZyklAktiv	:=
		IQ_stUniAnstgHMI.stMeldAusgHMI.bMeldEinlZyklBeendet:= FALSE;
		IQ_stUniAnstgHMI.stMeldAusgHMI.bMeldWarmlaufZykl	:= TRUE;
	ELSE							
		IQ_stUniAnstgHMI.stMeldAusgHMI.bMeldEinlZyklAktiv	:=
		IQ_stUniAnstgHMI.stMeldAusgHMI.bMeldEinlZyklBeendet:=
		IQ_stUniAnstgHMI.stMeldAusgHMI.bMeldWarmlaufZykl	:= FALSE;
	END_IF
END_ACTION

END_FUNCTION_BLOCK

// POUs/UniBausteine/FB_UniHydrAnstgHubb
///
///Beschreibung :	Allg. Ausgangsansteuerung (.Net-Vers.)
///					inkl. Händling - Handfkt.-Listen
///										- Meldfkt.-Listen
///										- Betriebsarten
///										- Schutzbereiche
///					Datentypen: Struct_UniBaustein
///									Struct_HandFktHMI
///					Ressourcen: GlobalVar_Allgemein
///									GlobalVar_AnlagHMI
///TwinCat Vers.:	3.1.4022.16							
///Erstellt		 :	B. Edenfeld (BECKHOFF AUTOMATION)
FUNCTION_BLOCK FB_UniHydrAnstgHubb
VAR_INPUT

	I_sStatName			:Tc2_System.T_MaxString;	// Aktueller Stationsname
	I_sAktorName		:Tc2_System.T_MaxString;	// Aktueller Aktorname von der Funktion des Aktors
	I_sAktorBMK1		:Tc2_System.T_MaxString;	// BMK - Rückmeldung

	I_bResHandFkt		: BOOL;							
	I_arrZuwGrdstFkt	: ARRAY[0..1] OF BOOL;		// Fkt.-Zuweisung Grdstlg.-ablauf
	I_arrZuwAutomFkt	: ARRAY[0..1] OF BOOL;		// Fkt.-Zuweisung Automatikablauf
                                                
	I_bAbfrAbsgPump	: BOOL;							// Abfrage Motorschutzschalter
	{attribute 'hide' := ''}                        
	I_nSchutzBer		: INT;							// Schutzbereich => Betriebsart
	{attribute 'hide' := ''}                     
	I_bVerrHdFktO		: BOOL;							// Sperren Handfkt. Auf (Oben)
	{attribute 'hide' := ''}                        
	I_bVerrHdFktU		: BOOL;							// Sperren Handfkt. Ab  (Unten)
	{attribute 'hide' := ''}	                     
	I_bEndlHdFktO		: BOOL;							// Endlage Handfkt. Auf (Oben)
	{attribute 'hide' := ''}                        
	I_bEndlHdFktU		: BOOL;                    // Endlage Handfkt. Ab  (Unten)
	
	I_eAnstgDef			:E_AnstgArtUniAktr := eAktrAusEinschalt;	// Definition der Meldetexte und Anzeigetexte.

	I_stVarInfoBMK		:__SYSTEM.VAR_INFO;	// Optional: __VARINFO von einem Hardwareeingang. Kann I_sAktorBMK1 ersetzen. I_sAktorBMK1 ist aber dominant. Nicht im Aufruf verwenden => separate Zuweisung

END_VAR
VAR_IN_OUT
	
	IQ_stUniAnstgHMI	:ST_UniAktrAnstg;	// HMI-Strukturen
	
END_VAR

VAR_OUTPUT
	///Arrayunter.- überschreitung
	{attribute 'hide' := ''}
	Q_nAufrufFehl		: INT;		
	Q_bAnstNetzPump	: BOOL;		// Netzansteuerung Auf (Pumpe)
	Q_bAnstNetzVent	: BOOL;		// Netzansteuerung Ab  (Ventil)
	Q_bMeldAbsgPump	: BOOL;     // Meldung Pumpenabsicherung
END_VAR

VAR
	sTextHandFkt1		:ARRAY[0..1] OF STRING(20);				
	sTextHandFkt2		:ARRAY[0..1] OF STRING(20);					
	sTextHandFktX		:ARRAY[0..1] OF STRING(20);	// Zum Zwischenspeichern

	rtrigHandFkt0: R_TRIG;
	rtrigHandFkt1: R_TRIG;
	
	//Relevante Variablen zur Diagnose
	stUniAnstgFkt		:ST_UniBaustein;
END_VAR

	(*Uni.- Hydraulikansteuerung*)

	(**************************************************)	
	(*Aufruf-Bereichskontrolle*)

	IF I_nSchutzBer <= 0 OR I_nSchutzBer > cAnzSchutzBer
	THEN
		Q_nAufrufFehl:= 1;
		RETURN;
	ELSE
		Q_nAufrufFehl:= 0;
	END_IF

	(**************************************************)	
	(*Haendling Uni-Struktur*)

	a_Standard();

	(**************************************************)	
	(*Ausgänge zuweisen*)

	x_AusgZuw();
	
	(**************************************************)	
	(*Zustände anzeigen*)

	y_ZustAnzg();

	(**************************************************)	
	(*Meldungen ausgeben*)

	z_FehlMeld();
	
	(**************************************************)

ACTION a_Standard:
	(*Ansteuerungstyp "Standard" /z.B. Hubbühnen (Pumpe/Ventil)*)

	(*Verwendete Handzeilen = 1 (s.Beispiel)*)

   (*    "Softkey Links"    /       "Handfunktion"       /   "Softkey Rechts"   *)
	(*                                                                           *) 
	(*_______absenken________/-------- Hubbühne ----------/________anheben_______*)

	(*Zeile 1 /Softkey Links	:Funktion ein.-ausschalten /Richtg. Auf*)
	(*Zeile 1 /Softkey Rechts	:Funktion ein.-ausschalten /Richtg. Ab*)

	(*Hinweis:
	- Funktion wird durch "VerrHdFkt" gesperrt (z.B. Niveau-LS...)
	- Funktion wird durch "EndlHdFkt" zurückgenommen
	*)
	
	(**************************************************)	

	stUniAnstgFkt.bHandAnw0:= IQ_stUniAnstgHMI.stHandFktHMI[1].bySwitch > 0;
	stUniAnstgFkt.bHandAnw1:= IQ_stUniAnstgHMI.stHandFktHMI[2].bySwitch > 0;
	
	IF arrBetrartAutomAktiv[I_nSchutzBer]
		OR I_bResHandFkt
		THEN
			stUniAnstgFkt.arrHandFkt[0]:=
			stUniAnstgFkt.arrHandFkt[1]:= FALSE;
		ELSE
			IF NOT arrBetrartAutomSpeichn[I_nSchutzBer]
				THEN
					IF NOT arrGrdstlgBetrAktiv[I_nSchutzBer]
						THEN
							 rtrigHandFkt1 (CLK:= stUniAnstgFkt.bHandAnw1);
							 IF rtrigHandFkt1.Q THEN
								 stUniAnstgFkt.arrHandFkt[1]:= NOT stUniAnstgFkt.arrHandFkt[1];
							 END_IF
							 IF NOT arrBetrartHandAktiv[I_nSchutzBer]
								 OR stUniAnstgFkt.arrHandFkt[0]
								 OR I_bVerrHdFktO OR I_bEndlHdFktO THEN
								 stUniAnstgFkt.arrHandFkt[1]:= FALSE;
							 END_IF
	 
							 rtrigHandFkt0 (CLK:= stUniAnstgFkt.bHandAnw0);
							 IF rtrigHandFkt0.Q THEN
								 stUniAnstgFkt.arrHandFkt[0]:= NOT stUniAnstgFkt.arrHandFkt[0];
							 END_IF
							 IF NOT arrBetrartHandAktiv[I_nSchutzBer]
								 OR stUniAnstgFkt.arrHandFkt[1]
								 OR I_bVerrHdFktU OR I_bEndlHdFktU THEN
								 stUniAnstgFkt.arrHandFkt[0]:= FALSE;
							 END_IF
					END_IF
			END_IF
	END_IF

	IF arrBetrartHandAktiv[I_nSchutzBer]
		THEN
			stUniAnstgFkt.nHandStat:= 0;			(*Funktion freigegeben*)
			
			IF stUniAnstgFkt.arrHandFkt[1]
				THEN
					stUniAnstgFkt.nHandStat:= 2;	(*Funktion Rechts aktiv*)
			END_IF
			IF stUniAnstgFkt.arrHandFkt[0]
				THEN
					stUniAnstgFkt.nHandStat:= 1;	(*Funktion Links aktiv*)
			END_IF
		ELSE
			stUniAnstgFkt.nHandStat:= 256;		(*Funktion gesperrt*)
	END_IF

	(**************************************************)	

	IF arrBetrartHandAktiv[I_nSchutzBer]
		THEN
			stUniAnstgFkt.arrGrdstFkt[0]:= I_arrZuwGrdstFkt[0];
			stUniAnstgFkt.arrGrdstFkt[1]:= I_arrZuwGrdstFkt[1];
		ELSE
			stUniAnstgFkt.arrGrdstFkt[0]:= 
			stUniAnstgFkt.arrGrdstFkt[1]:= FALSE;
   END_IF
	IF arrBetrartAutomAktiv[I_nSchutzBer] OR TRUE //ToDo
		THEN
			stUniAnstgFkt.arrAutomFkt[0]:= I_arrZuwAutomFkt[0];
			stUniAnstgFkt.arrAutomFkt[1]:= I_arrZuwAutomFkt[1];
		ELSE
			stUniAnstgFkt.arrAutomFkt[0]:= 
			stUniAnstgFkt.arrAutomFkt[1]:= FALSE;
   END_IF

	(**************************************************)	

	stUniAnstgFkt.arrFktAusfg[0]:= stUniAnstgFkt.arrGrdstFkt[0]
											  OR stUniAnstgFkt.arrHandFkt[0]
											  OR stUniAnstgFkt.arrAutomFkt[0];

	stUniAnstgFkt.arrFktAusfg[1]:= stUniAnstgFkt.arrGrdstFkt[1]
											  OR stUniAnstgFkt.arrHandFkt[1]
											  OR stUniAnstgFkt.arrAutomFkt[1];

	(**************************************************)
END_ACTION

ACTION x_AusgZuw:
	
	(**************************************************)	
	(*Ausgänge zuweisen*)

	Q_bAnstNetzPump:= stUniAnstgFkt.arrFktAusfg[1]
						 	AND NOT Q_bAnstNetzVent
						 	AND arrAntrGruppeFrg[I_nSchutzBer]
						 	AND I_bAbfrAbsgPump
						 	AND bVersEingAusgSchaltsOk;

	Q_bAnstNetzVent:= stUniAnstgFkt.arrFktAusfg[0]
						 	AND NOT Q_bAnstNetzPump
						 	AND arrAntrGruppeFrg[I_nSchutzBer]
						 	AND bVersEingAusgSchaltsOk;
END_ACTION

ACTION y_ZustAnzg:
	
	(**************************************************)	
	(*Zustände anzeigen*)
	CASE I_eAnstgDef OF 
eAktrAusEinschalt,
eAktrEinAusschalt:
						sTextHandFkt1[0]:= 'einschalten';
						sTextHandFkt1[1]:= 'eingeschaltet';
						sTextHandFkt2[0]:= 'ausschalten';
						sTextHandFkt2[1]:= 'ausgeschaltet';
eAktrAusEinfahr,
eAktrEinAusfahr:
						sTextHandFkt1[0]:= 'einfahren';
						sTextHandFkt1[1]:= 'eingefahren';
						sTextHandFkt2[0]:= 'ausfahren';
						sTextHandFkt2[1]:= 'ausgefahren';
eAktrHebenSenken,
eAktrSenkenHeben:
						sTextHandFkt1[0]:= 'senken';
						sTextHandFkt1[1]:= 'abgesenkt';
						sTextHandFkt2[0]:= 'heben';
						sTextHandFkt2[1]:= 'angehoben';
	END_CASE
	
	IF I_eAnstgDef >= 20 //Zuweisungen tauschen 
		THEN
			sTextHandFktX:= sTextHandFkt1; 
			sTextHandFkt1:= sTextHandFkt2;
			sTextHandFkt2:= sTextHandFktX;
	END_IF
	
	IF stUniAnstgFkt.nHandStat = 1	(*Handfunktion.1 aktiv*)
		THEN
			IQ_stUniAnstgHMI.stHandFktHMI[1].sColour:= cGruenAsString;
			IQ_stUniAnstgHMI.stHandFktHMI[1].sText:= sTextHandFkt1[1];
		ELSE
			IQ_stUniAnstgHMI.stHandFktHMI[1].sColour:= cDefaultAsString;
			IQ_stUniAnstgHMI.stHandFktHMI[1].sText:= sTextHandFkt1[0];
   END_IF
	IF stUniAnstgFkt.nHandStat = 2	(*Handfunktion.2 aktiv*)
		THEN		 
			IQ_stUniAnstgHMI.stHandFktHMI[2].sColour:= cGruenAsString;
			IQ_stUniAnstgHMI.stHandFktHMI[2].sText:= sTextHandFkt2[1];
		ELSE
			IQ_stUniAnstgHMI.stHandFktHMI[2].sColour:= cDefaultAsString;
			IQ_stUniAnstgHMI.stHandFktHMI[2].sText:= sTextHandFkt2[0];
   END_IF
	IF stUniAnstgFkt.nHandStat = 256	(*Funktion gesperrt*)
		THEN
			IQ_stUniAnstgHMI.stHandFktHMI[1].byStatus:=
			IQ_stUniAnstgHMI.stHandFktHMI[2].byStatus:= 1;
			IQ_stUniAnstgHMI.stHandFktHMI[1].sText:= sTextHandFkt1[0];
			IQ_stUniAnstgHMI.stHandFktHMI[2].sText:= sTextHandFkt2[0];
		ELSE
			IQ_stUniAnstgHMI.stHandFktHMI[1].byStatus:=
			IQ_stUniAnstgHMI.stHandFktHMI[2].byStatus:= 0;
   END_IF

	(**************************************************)
END_ACTION

ACTION z_FehlMeld:

	(**************************************************)	
	(*Meldungen ausgeben*)

	Q_bMeldAbsgPump:= arrAntrGruppeFrg[I_nSchutzBer]
							AND NOT I_bAbfrAbsgPump
							AND bVersEingAusgSchaltsOk;
		
	IQ_stUniAnstgHMI.stMeldAusgHMI.SourceID			:= 0;	// Nicht mehr verwendet
	IQ_stUniAnstgHMI.stMeldAusgHMI.SourceName			:= I_sStatName;
	IQ_stUniAnstgHMI.stMeldAusgHMI.sAktorName			:= I_sAktorName;
	
	IF I_sAktorBMK1 <> ''
	THEN	// I_sAktorBMK1 ist beschrieben. Damit wird der String als BMK genommen
		IQ_stUniAnstgHMI.stMeldAusgHMI.sBMK	:= I_sAktorBMK1;
	ELSE	// Der Kommentar von VARINFO wird als BMK genommen
		IQ_stUniAnstgHMI.stMeldAusgHMI.sBMK	:= I_stVarInfoBMK.Comment;
	END_IF

	IQ_stUniAnstgHMI.stMeldAusgHMI.bLfzMeldAusg		:= Q_bMeldAbsgPump
																		OR bTestMeldAktr; 
	IQ_stUniAnstgHMI.stMeldAusgHMI.bMeldHinweis		:= FALSE;	

		
	(**************************************************)
END_ACTION

END_FUNCTION_BLOCK

// POUs/UniBausteine/FB_UniWkzgAnstg
(*
Beschreibung :	UniFB zur Hardwaresteuerung, Anzeige und Fehlermeldung in der Avalon HMI eines Werkzeuges ohne zustandsabfragen Abfragen.
					inkl. Handling - Handfunktinen
										- Meldefunktionen
										- Betriebsarten
										- Schutzbereiche
					Datentypen: ST_UniBaustein
									ST_UniWkzgAnstg
					Ressourcen: GlobalVar_Allgemein
									GlobalVar_Farben
									AllgemeineParameter
TwinCat Vers.:	3.1.4024.25							
Erstellt		 :	Anlagentechnik Grp.11 (BECKHOFF AUTOMATION)
*)
FUNCTION_BLOCK FB_UniWkzgAnstg
VAR_INPUT

	I_sStatName			:Tc2_System.T_MaxString;	// Aktueller Stationsname
	I_sAktorName		:Tc2_System.T_MaxString;	// Aktuelles Werkzeugs von der Funktion des Werkzeuges
	
	I_bResHandFkt		:BOOL;	// Funktion-Reset für Grundstellungsablauf
	I_bZuwGrdstFkt		:BOOL;	// Funktion-Zuweisung Grundstellungsablauf
	I_bZuwAutomFkt		:BOOL;	// Funktion-Zuweisung Automatikablauf
																						
	I_sZuDef0			:Tc2_System.T_MaxString;	// eigene Definition für die linke Tasterbeschriftung
	I_sInDef0			:Tc2_System.T_MaxString;	// eigene Definition für die linke Tasterbeschriftung
	I_sZuDef1			:Tc2_System.T_MaxString;	// eigene Definition für die rechte Tasterbeschriftung
	I_sInDef1			:Tc2_System.T_MaxString;	// eigene Definition für die rechte Tasterbeschriftung
	I_eAnstgDef			:E_AnstgArtUniWkzg;		(*Definition Ansteuerung*)
										(*1: Funktionstext: Grd.-Arbeitsstlg.*)
										(*2:       "      : Abs.-Anheben*)
										(*3:       "      : Ein.-Ausfahren*) 
										(*4:       "      : Zur.-Vorfahren*) 
										(*5:       "      : Ein.-Aussteuern*) 
										(*6:       "      : Loes.-Spannen*) 
										(*7:       "      : Oeffn.-Greifen*)
										(*8:       "      : Klemm.-Loesen*) 

	I_nSchutzBer		:INT;		(*Schutzbereich => Betriebsart*)

	(*Optionale Funktionen*)													
	I_bResHdBetr		:BOOL;	(*Zurücksetzen bei Handbetrieb*)
																					
	I_tHdPulsVorg		:TIME;	(*Max. Handfkt.-Ansteuerdauer*)
																					
	I_bAnstgUng			:BOOL;	(*Ansteuerung Ungeschaltet*)		
	I_bAnstgInvt		:BOOL;	(*Ansteuerung Invertieren*)

END_VAR
VAR_IN_OUT
																						
	IQ_stUniAnstgHMI	:ST_UniWkzgAnstg;	(*HMI-Strukturen*)
																						
END_VAR
VAR_OUTPUT
												
	Q_bWkzgAnstg		:BOOL;	(*Ansteuerung Arbeitsstellung*)

END_VAR
VAR
																					
	tpHdPulsUebw		:TP;
																						
	bHdPulsAnstg		:BOOL;													
																					
	sTextHandFkt1		:ARRAY[0..1] OF STRING(20);						
	sTextHandFkt2		:ARRAY[0..1] OF STRING(20);						
	sTextHandFktX		:ARRAY[0..1] OF STRING(20);	// Wird für den Vertausch der Texte benötigt.
	
	//Relevante Variablen zur Diagnose
	stUniAnstgFkt		:ST_UniBaustein;

END_VAR

	(*Uni.- Werkzeugansteuerung*)
	
	(**************************************************)	
	(*Aufruf-Bereichskontrolle*)

	IF I_nSchutzBer <= 0 OR I_nSchutzBer > cAnzSchutzBer
	THEN
		IQ_stUniAnstgHMI.stMeldAusgHMI.sMeldText		:= 'I_nSchutzBer = 0 oder zu gross.';
		IQ_stUniAnstgHMI.stMeldAusgHMI.bMeldHinweis	:= TRUE;
			
		stUniAnstgFkt.nHandStat:= 256;	// Funktion sperren
		y_ZustAnzg();
		RETURN;
	ELSE
		IQ_stUniAnstgHMI.stMeldAusgHMI.bMeldHinweis	:= FALSE;
		IQ_stUniAnstgHMI.stMeldAusgHMI.sMeldText		:= '';
	END_IF

	(**************************************************)	
	(*Haendling Uni-Struktur*)

	bHdPulsAnstg:= TIME_TO_BOOL(I_tHdPulsVorg);
	
	IF NOT bHdPulsAnstg
		THEN	
			a_Standard();
		ELSE	 
			b_PulsUebw();
   END_IF

	(**************************************************)	
	(*Ausgänge zuweisen*)

	x_AusgZuw();
	
	(**************************************************)	
	(*Zustände anzeigen*)

	y_ZustAnzg();

	(**************************************************)	
	(*Meldungen ausgeben*)

	z_FehlMeld();
	
	(**************************************************)

ACTION a_Standard:
	(*Ansteuerungstyp "Standard" /z.B. Bohrspindeln...*)

	(*Verwendete Softkeytasten = 2 (s.Beispiel)*)

   (*       "Handfunktion"       /   "Softkeytaste 1"   /   "Softkeytaste 2"   *)
	(*                                                                          *) 
   (*-------- Bohrspindel -------/______einsteuern______/______aussteuern______*)
	
	(*Softkeyleiste.1		:Funktion ausschalten*)
	(*Softkeyleiste.2		:Funktion einschalten*)

	(*Hinweis:
	- Funktion wird durch "ResHdBetr" bei Betriebsartenwechsel zurückgenommen
	
	- Bei "AnstgUng" bleiben die F-Ausgänge auch bei geöffn. Schutzbereich aktiv  
	- Bei "AnstgInvt" wird die Logik der Funktions-Ausgänge invertiert  
	*)

	(**************************************************)	

	stUniAnstgFkt.bHandAnw0:= IQ_stUniAnstgHMI.stHandFktHMI[1].bySwitch > 0;
	stUniAnstgFkt.bHandAnw1:= IQ_stUniAnstgHMI.stHandFktHMI[2].bySwitch > 0;
	
	IF arrBetrartAutomAktiv[I_nSchutzBer]
		OR I_bResHandFkt
		THEN
			stUniAnstgFkt.arrHandFkt[1]:= FALSE;
		ELSE
			IF arrBetrartAutomSpeichn[I_nSchutzBer]
				THEN
					IF NOT I_bResHdBetr THEN
						stUniAnstgFkt.arrHandFkt[1]:= stUniAnstgFkt.arrFktAusfg[1];
					END_IF
				ELSE
					IF NOT arrGrdstlgBetrAktiv[I_nSchutzBer]
						AND arrBetrartHandAktiv[I_nSchutzBer]
						THEN
							 IF stUniAnstgFkt.bHandAnw1 THEN
								 stUniAnstgFkt.arrHandFkt[1]:= TRUE;
							 END_IF
							 IF stUniAnstgFkt.bHandAnw0 THEN
								 stUniAnstgFkt.arrHandFkt[1]:= FALSE;
							 END_IF
					END_IF
			END_IF
	END_IF

	IF arrBetrartHandAktiv[I_nSchutzBer]
		THEN
			IF stUniAnstgFkt.arrHandFkt[1]
				THEN
					stUniAnstgFkt.nHandStat:= 2;	(*Handfunktion.2 aktiv*)
				ELSE
					stUniAnstgFkt.nHandStat:= 1;	(*Handfunktion.1 aktiv*)
			END_IF
		ELSE
			stUniAnstgFkt.nHandStat:= 256;		(*Funktion gesperrt*)
	END_IF

	(**************************************************)	

	IF arrBetrartHandAktiv[I_nSchutzBer]
		THEN
			stUniAnstgFkt.arrGrdstFkt[1]:= I_bZuwGrdstFkt;
		ELSE
			stUniAnstgFkt.arrGrdstFkt[1]:= FALSE;
   END_IF
	IF arrBetrartAutomAktiv[I_nSchutzBer] OR TRUE //ToDo
		THEN
			stUniAnstgFkt.arrAutomFkt[1]:= I_bZuwAutomFkt;
		ELSE
			stUniAnstgFkt.arrAutomFkt[1]:= FALSE;
   END_IF

	(**************************************************)	

	stUniAnstgFkt.arrFktAusfg[1]:= stUniAnstgFkt.arrGrdstFkt[1]
										  	 OR stUniAnstgFkt.arrHandFkt[1]
										    OR stUniAnstgFkt.arrAutomFkt[1];

	(**************************************************)
END_ACTION

ACTION b_PulsUebw:
	(*Ansteuerungstyp "Pulsüberwachg." /z.B. Leimdüsen...*)

	(*Verwendete Softkeytasten = 2 (s.Beispiel)*)

   (*       "Handfunktion"       /   "Softkeytaste 1"   /   "Softkeytaste 2"   *)
	(*                                                                          *) 
   (*-------- Leimdüse 01 -------/_________aus__________/_________ein__________*)
	
	(*Softkeyleiste.1		:Funktion ausschalten*)
	(*Softkeyleiste.2		:Funktion einschalten*)

	(*Hinweis:
	- Mit "HdPulsVorg" kann die Max. Handfunktionsdauer begrenzt werden
	
	- Bei "AnstgUng" bleiben die F-Ausgänge auch bei geöffn. Schutzbereich aktiv  
	- Bei "AnstgInvt" wird die Logik der Funktions-Ausgänge invertiert  
	*)

	(**************************************************)	

	stUniAnstgFkt.bHandAnw0:= IQ_stUniAnstgHMI.stHandFktHMI[1].bySwitch > 0;
	stUniAnstgFkt.bHandAnw1:= IQ_stUniAnstgHMI.stHandFktHMI[2].bySwitch > 0;
	
	IF arrBetrartAutomAktiv[I_nSchutzBer]
		OR I_bResHandFkt
		THEN
			stUniAnstgFkt.arrHandFkt[1]:= FALSE;
		ELSE
			IF NOT arrBetrartAutomSpeichn[I_nSchutzBer]
				THEN
					IF NOT arrGrdstlgBetrAktiv[I_nSchutzBer]
						THEN
							tpHdPulsUebw (IN:= stUniAnstgFkt.bHandAnw1,
								 			  PT:= I_tHdPulsVorg,
											  Q => stUniAnstgFkt.arrHandFkt[1]);		
							IF NOT arrBetrartHandAktiv[I_nSchutzBer]
							   OR stUniAnstgFkt.bHandAnw0 THEN
								stUniAnstgFkt.arrHandFkt[1]:= FALSE;
							END_IF
					END_IF
			END_IF
	END_IF

	IF arrBetrartHandAktiv[I_nSchutzBer]
		THEN
			IF stUniAnstgFkt.arrHandFkt[1]
				THEN
					stUniAnstgFkt.nHandStat:= 2;	(*Handfunktion.2 aktiv*)
				ELSE
					stUniAnstgFkt.nHandStat:= 1;	(*Handfunktion.1 aktiv*)
			END_IF
		ELSE
			stUniAnstgFkt.nHandStat:= 256;		(*Funktion gesperrt*)
	END_IF

	(**************************************************)	

	IF arrBetrartHandAktiv[I_nSchutzBer]
		THEN
			stUniAnstgFkt.arrGrdstFkt[1]:= I_bZuwGrdstFkt;
		ELSE
			stUniAnstgFkt.arrGrdstFkt[1]:= FALSE;
   END_IF
	IF arrBetrartAutomAktiv[I_nSchutzBer] OR TRUE //ToDo
		THEN
			stUniAnstgFkt.arrAutomFkt[1]:= I_bZuwAutomFkt;
		ELSE
			stUniAnstgFkt.arrAutomFkt[1]:= FALSE;
   END_IF

	(**************************************************)	

	stUniAnstgFkt.arrFktAusfg[1]:= stUniAnstgFkt.arrGrdstFkt[1]
										  	 OR stUniAnstgFkt.arrHandFkt[1]
										    OR stUniAnstgFkt.arrAutomFkt[1];

	(**************************************************)
END_ACTION

ACTION x_AusgZuw:

	(**************************************************)	
	(*Ausgänge zuweisen*)

	Q_bWkzgAnstg:= stUniAnstgFkt.arrFktAusfg[1]
					 	AND (arrAusgGruppeFrg[I_nSchutzBer]
				    	OR I_bAnstgUng)
					 	AND bVersEingAusgAnlagOk;

	(**************************************************)	
	(*Ausgänge invertieren*)

	IF I_bAnstgInvt THEN
		Q_bWkzgAnstg:= NOT Q_bWkzgAnstg;
	END_IF

	(**************************************************)
END_ACTION

ACTION y_ZustAnzg:
	
	(**************************************************)	
	(*Zustände anzeigen*)

// die Zahlen 0-8 sind wegen der Abwärtskompatibiliät noch drin.
CASE I_eAnstgDef OF
	
0,eWkzgDef0Def1,eWkzgDef1Def0:
	sTextHandFkt1[0]:= I_sZuDef0;
	sTextHandFkt1[1]:= I_sInDef0;
	sTextHandFkt2[0]:= I_sZuDef1;
	sTextHandFkt2[1]:= I_sInDef1;
1,eWkzgGrdArbstlg,eWkzgArbGrdstlg:
	sTextHandFkt1[0]:= 'zur Grundstlg.';
	sTextHandFkt1[1]:= 'in Grundstlg.';
	sTextHandFkt2[0]:= 'zur Arbeitstlg.';
	sTextHandFkt2[1]:= 'in Arbeitstlg.';
2,eWkzgAbsAnheb,eWkzgAnhAbsenk:
	sTextHandFkt1[0]:= 'absenken';
	sTextHandFkt1[1]:= 'abgesenkt';
	sTextHandFkt2[0]:= 'anheben';
	sTextHandFkt2[1]:= 'angehoben';
3,eWkzgEinAusfahr,eWkzgAusEinfahr:
	sTextHandFkt1[0]:= 'einfahren';
	sTextHandFkt1[1]:= 'eingefahren';
	sTextHandFkt2[0]:= 'ausfahren';
	sTextHandFkt2[1]:= 'ausgefahren';
4,eWkzgZurVorfahr,eWkzgVorZurfahr:
	sTextHandFkt1[0]:= 'zurückfahren';
	sTextHandFkt1[1]:= 'zurückgefahren';
	sTextHandFkt2[0]:= 'vorfahren';
	sTextHandFkt2[1]:= 'vorgefahren';
5,eWkzgEinAussteun,eWkzgAusEinsteun:
	sTextHandFkt1[0]:= 'einsteuern';
	sTextHandFkt1[1]:= 'eingesteuert';
	sTextHandFkt2[0]:= 'aussteuern';
	sTextHandFkt2[1]:= 'ausgesteuert';
6,eWkzgLoesSpann,eWkzgSpannLoes:
	sTextHandFkt1[0]:= 'lösen';
	sTextHandFkt1[1]:= 'gelöst';
	sTextHandFkt2[0]:= 'spannen';
	sTextHandFkt2[1]:= 'gespannt';
7,eWkzgOeffnSchliess,eWkzgSchliessOeffn:
	sTextHandFkt1[0]:= 'öffnen';
	sTextHandFkt1[1]:= 'geöffnet';
	sTextHandFkt2[0]:= 'schliessen';
	sTextHandFkt2[1]:= 'geschlossen';
8,eWkzgKlemLoesen,eWkzgLoesKlem:
	sTextHandFkt1[0]:= 'klemmen';
	sTextHandFkt1[1]:= 'geklemmt';
	sTextHandFkt2[0]:= 'lösen';
	sTextHandFkt2[1]:= 'gelöst';
END_CASE 
	
	IF I_eAnstgDef >= 50 //Zuweisungen tauschen 
		THEN
			sTextHandFktX:= sTextHandFkt1; 
			sTextHandFkt1:= sTextHandFkt2;
			sTextHandFkt2:= sTextHandFktX;
	END_IF
	
	IF stUniAnstgFkt.nHandStat = 1	(*Handfunktion.1 aktiv*)
		THEN
			IQ_stUniAnstgHMI.stHandFktHMI[1].sColour:= cGruenAsString;
			IQ_stUniAnstgHMI.stHandFktHMI[1].sText:= sTextHandFkt1[1];
		ELSE
			IQ_stUniAnstgHMI.stHandFktHMI[1].sColour:= cDefaultAsString;
			IQ_stUniAnstgHMI.stHandFktHMI[1].sText:= sTextHandFkt1[0];
   END_IF
	IF stUniAnstgFkt.nHandStat = 2	(*Handfunktion.2 aktiv*)
		THEN		 
			IQ_stUniAnstgHMI.stHandFktHMI[2].sColour:= cGruenAsString;
			IQ_stUniAnstgHMI.stHandFktHMI[2].sText:= sTextHandFkt2[1];
		ELSE
			IQ_stUniAnstgHMI.stHandFktHMI[2].sColour:= cDefaultAsString;
			IQ_stUniAnstgHMI.stHandFktHMI[2].sText:= sTextHandFkt2[0];
   END_IF
	IF stUniAnstgFkt.nHandStat = 256	(*Funktion gesperrt*)
		THEN
			IQ_stUniAnstgHMI.stHandFktHMI[1].byStatus:=
			IQ_stUniAnstgHMI.stHandFktHMI[2].byStatus:= 1;
		ELSE
			IQ_stUniAnstgHMI.stHandFktHMI[1].byStatus:=
			IQ_stUniAnstgHMI.stHandFktHMI[2].byStatus:= 0;
   END_IF

	(**************************************************)
END_ACTION

ACTION z_FehlMeld:

	(**************************************************)	
	(*Meldungen ausgeben*)

	//Uni-Ansteuerung ohne Meldungen

	(**************************************************)
END_ACTION

END_FUNCTION_BLOCK

// POUs/UniBausteine/FB_UniZyliAnstg
(*
Beschreibung :	UniFB zur Hardwaresteuerung, Anzeige und Fehlermeldung in der Avalon HMI eines allgemeinen Ventil mit Zylinders mit Testmodus zum Reversieren
					inkl. Handling - Handfunktinen
										- Meldefunktionen
										- Betriebsarten
										- Schutzbereiche
					Datentypen: ST_UniBaustein
									ST_UniZyliAnstg_TestMode
					Ressourcen: GlobalVar_Allgemein
									GlobalVar_Farben
									AllgemeineParameter
TwinCat Vers.:	3.1.4024.25							
Erstellt		 :	Anlagentechnik Grp.11 (BECKHOFF AUTOMATION)
*)
FUNCTION_BLOCK FB_UniZyliAnstg
VAR_INPUT

	I_sStatName			:Tc2_System.T_MaxString;	// Aktueller Stationsname
	I_sAktorName		:Tc2_System.T_MaxString;	// Aktueller Zylindername mit der Funktion des Zylinder
	I_sAktorBMK0		:Tc2_System.T_MaxString;	// BMK - Ruhestellung
	I_sAktorBMK1		:Tc2_System.T_MaxString;	// BMK - Arbeitsstellung

	I_bResHandFkt		:BOOL;						// Funktion-Reset für Grundstellungsablauf
	I_arrZuwGrdstFkt	:ARRAY[0..1] OF BOOL;	// Funktion-Zuweisung Grundstellungsablauf
	I_arrZuwAutomFkt	:ARRAY[0..1] OF BOOL;	// Funktion-Zuweisung Automatikablauf

	I_bZyliAbfrg0		:BOOL;	// Abfrage Ruhestellung
	I_bZyliAbfrg1		:BOOL;	// Abfrage Arbeitsstellung

	I_sZuDef0			:Tc2_System.T_MaxString;	// eigene Definition für die linke Tasterbeschriftung
	I_sInDef0			:Tc2_System.T_MaxString;	// eigene Definition für die linke Tasterbeschriftung
	I_sZuDef1			:Tc2_System.T_MaxString;	// eigene Definition für die rechte Tasterbeschriftung
	I_sInDef1			:Tc2_System.T_MaxString;	// eigene Definition für die rechte Tasterbeschriftung
	I_sLzFehlerDef0	:Tc2_System.T_MaxString;	// Laufzeitfehler wenn nicht in Def0
	I_sLzFehlerDef1	:Tc2_System.T_MaxString;	// Laufzeitfehler wenn nicht in Def1
	I_sSensorFehlDef	:Tc2_System.T_MaxString;	// Sensorfehelr wenn nicht in Def0 oder Def1

	I_eAnstgDef			:E_AnstgArtUniZyli;		// Definition Ansteuerung
										// 10: Funktionstext: Definition0 - Def1
										// 11:			"		 : Grd.-Arbeitsstlg.
										// 12:       "		 : Abs.-Anheben
										// 13:       "      : Ein.-Ausfahren 
										// 14:       "      : Zur.-Vorfahren 
										// 15:       "      : Ein.-Aussteuern 
										// 16:       "      : Loes.-Spannen 
										// 17:       "      : Oeffn.-Greifen 

	I_eAnstgTyp			:E_ZylinderTyp;	// Eingesetzter Zylindertyp
										// 1: Anstg. 1 Rückstlg. /Abfrg.0
								   	// 2: Anstg. 1 Rückstlg. /Abfrg.0-1
								   	// 3: Anstg. 0-1 Rückstlg. /Abfrg.0
								   	// 4: Anstg. 0-1 Rückstlg. /Abfrg.0-1
								   	// 5: Anstg. 0-1 Impulsstlg. /Abfrg.0
								   	// 6: Anstg. 0-1 Impulsstlg. /Abfrg.0-1
								   	// 7: Anstg. 0-1 Mittelstlg. /Abfrg.0-1

	I_nSchutzBer		:INT;		// Schutzbereich => Betriebsart	

	// Optionale Funktionen													
	I_bResHdBetr		:BOOL;	// Zurücksetzen der Ventilansteuerung beim Wechsel auf Handbetrieb

	I_bVerrHdFkt0		:BOOL;	// Sperren Handfunktionen Ruhestellung
	I_bVerrHdFkt1		:BOOL;	// Sperren Handfunktionen Arbeitsstellung

	I_tLaufzVorg		:TIME:= T#5S;	// Meldelaufzeit
	I_bVerrMeldg		:BOOL;	// Meldungsausgabe allgemein unterdrücken
	I_bVerrMeldg0		:BOOL;	// nur Meldung für die Ansteuerung 0 unterdrücken
	I_bVerrMeldg1		:BOOL;	// nur Meldung für die Ansteuerung 1 unterdrücken

	I_bAnstgUntbr		:BOOL;	// Ansteuerung Unterbrechen		
	I_bAnstgUng			:BOOL;	// Ansteuerung Ungeschaltet		
	I_bAnstgInvt		:BOOL;	// Ansteuerung Invertieren

	I_stVarInfoBMK0	:__SYSTEM.VAR_INFO;	// Optional: __VARINFO von dem Hardwareeingang I_bZyliAbfrg0. Kann I_sAktorBMK0 ersetzen. I_sAktorBMK0 ist aber dominant. Nicht im Aufruf verwenden => separate Zuweisung
	I_stVarInfoBMK1	:__SYSTEM.VAR_INFO;	// Optional: __VARINFO von dem Hardwareeingang I_bZyliAbfrg1. Kann I_sAktorBMK1 ersetzen. I_sAktorBMK1 ist aber dominant. Nicht im Aufruf verwenden => separate Zuweisung
END_VAR
VAR_IN_OUT

	IQ_stUniAnstgHMI	:ST_UniZyliAnstg;	// HMI-Strukturen

END_VAR
VAR_OUTPUT

	Q_bZyliAnstg0		:BOOL;	// Ansteuerung Ruhestellung
	Q_bZyliAnstg1		:BOOL;	// Ansteuerung Arbeitsstellung

END_VAR
VAR

	sTextHandFkt1		:ARRAY[0..1] OF STRING(20);					
	sTextHandFkt2		:ARRAY[0..1] OF STRING(20);					
	sTextHandFktX		:ARRAY[0..1] OF STRING(20);	

	fbLfzMeldAusg		:FB_LaufzMeldg;
	bLaufzMeldg0		:BOOL;
	bLaufzMeldg1		:BOOL;
	
	// TestMode zum Reversieren des Zylinders
	bTestModeAktiv		:BOOL;	// Merker für den Testmode
	rTrigTestMode		:Tc2_Standard.R_TRIG;	// Trigger für Testmode
	tReversierZeit		:TIME;	// Reversierzeit im Testmode
	fbReversierTakt	:FB_Blinker;	// Reversiertakt erzeugen
	rTrigEndlage0		:Tc2_Standard.R_TRIG;	// Zur Zeitmessung bis in Endlage0
	rTrigEndlage1		:Tc2_Standard.R_TRIG;	// Zur Zeitmessung bis in Endlage0
	tBisInEndlage0		:TIME;	// Gemessene Zeit bis in Endlage0
	tBisInEndlage1		:TIME;	// Gemessene Zeit bis in Endlage1

	//Relevante Variablen zur Diagnose
	stUniAnstgFkt		:ST_UniBaustein;
END_VAR

//****************************************************************************************************
// Uni - Zylinderansteuerung
//****************************************************************************************************
	
// Aufruf-Bereichskontrolle

IF I_nSchutzBer = 0 OR I_nSchutzBer > cAnzSchutzBer
THEN
	IQ_stUniAnstgHMI.stMeldAusgHMI.sMeldText		:= 'I_nSchutzBer = 0 oder zu gross.';
	IQ_stUniAnstgHMI.stMeldAusgHMI.SourceName		:= I_sStatName;
	IQ_stUniAnstgHMI.stMeldAusgHMI.sAktorName		:= I_sAktorName;
	IQ_stUniAnstgHMI.stMeldAusgHMI.bMeldHinweis	:= TRUE;
	stUniAnstgFkt.nHandStat:= 256;	// Funktion sperren
	y_ZustaendeAnzeigen();
	RETURN;
ELSE
	IQ_stUniAnstgHMI.stMeldAusgHMI.bMeldHinweis	:= FALSE;
	IQ_stUniAnstgHMI.stMeldAusgHMI.sMeldText		:= '';
END_IF

//****************************************************************************************************
// Haendling Uni-Struktur

CASE I_eAnstgTyp OF

1..6:	// Zylindertyp Standard

	a_Standard();

7:		// Zylindertyp Mittelstellung	

	b_MittelStellung();

END_CASE


//****************************************************************************************************
// Testmode

c_TestMode();

//****************************************************************************************************
// Ausgänge zuweisen

x_AusgaengeZuweisen();
	
//****************************************************************************************************
// Zustände anzeigen

y_ZustaendeAnzeigen();

//****************************************************************************************************
// Meldungen ausgeben

z_FehlerMeldung();
	
//****************************************************************************************************

ACTION a_Standard:
//****************************************************************************************************
	// Ansteuerungstyp "Standard" /Allgemeine Standardpneumatikzylinder...

	// Verwendete Softkeytasten = 2 (s.Beispiel)

   (*       "Handfunktion"       /   "Softkeytaste 1"   /   "Softkeytaste 2"   *)
	(*                                                                          *) 
	(*------- Stopanschlag -------/_______absenken_______/_______anheben________*)
	
	(*Softkeyleiste.1		:Funktion ausschalten*)
	(*Softkeyleiste.2		:Funktion einschalten*)

	(*Hinweis:
	- Funktion wird durch "ResHdBetr" bei Betriebsartenwechsel zurückgenommen
	- Funktion wird durch "VerrHdFkt" gesperrt (z.B. bei Kollissionserkennung...)
	
	- Mit "LaufzVorg" kann die Meldelaufzeit angepasst werden (Default: 5sek)
	- Mit "VerrMeldg" wird die Meldeausgabe unterdrückt (eventl. Ablaufbedingt)
	
	- Bei "AnstgUntbr" werden die F-Ausgänge deaktiviert (z.B. bei LSG-Unterbr.)
				         Erforderlich u.U. bei Sonderbeschaltung einzelner Ausgänge
	- Bei "AnstgUng" bleiben die F-Ausgänge auch bei geöffn. Schutzbereich aktiv  
	- Bei "AnstgInvt" wird die Logik der Funktions-Ausgänge invertiert  
	*)

//****************************************************************************************************

stUniAnstgFkt.bHandAnw0:= IQ_stUniAnstgHMI.stHandFktHMI[1].bySwitch > 0;
stUniAnstgFkt.bHandAnw1:= IQ_stUniAnstgHMI.stHandFktHMI[2].bySwitch > 0;

IF arrBetrartAutomAktiv[I_nSchutzBer]
	OR I_bResHandFkt
THEN
	stUniAnstgFkt.arrHandFkt[1]:= FALSE;
ELSE
	IF arrBetrartAutomSpeichn[I_nSchutzBer]
	THEN
		IF NOT I_bResHdBetr
		THEN
			stUniAnstgFkt.arrHandFkt[1]:= stUniAnstgFkt.arrFktAusfg[1];
		END_IF
	ELSE
		IF (NOT arrGrdstlgBetrAktiv[I_nSchutzBer]
				AND arrBetrartHandAktiv[I_nSchutzBer])
			OR I_bAnstgUng
		THEN
			IF stUniAnstgFkt.bHandAnw1
				AND NOT I_bVerrHdFkt1
			THEN
				 stUniAnstgFkt.arrHandFkt[1]:= TRUE;
			END_IF
			IF stUniAnstgFkt.bHandAnw0
				AND NOT I_bVerrHdFkt0
			THEN
				stUniAnstgFkt.arrHandFkt[1]:= FALSE;
			END_IF
		END_IF
	END_IF
END_IF

//****************************************************************************************************

IF arrBetrartHandAktiv[I_nSchutzBer]
	THEN
		stUniAnstgFkt.arrGrdstFkt[1]:= I_arrZuwGrdstFkt[1];
	ELSE
		stUniAnstgFkt.arrGrdstFkt[1]:= FALSE;
END_IF
IF arrBetrartAutomAktiv[I_nSchutzBer] OR TRUE //ToDo
	THEN
		stUniAnstgFkt.arrAutomFkt[1]:= I_arrZuwAutomFkt[1];
	ELSE
		stUniAnstgFkt.arrAutomFkt[1]:= FALSE;
END_IF

//****************************************************************************************************

stUniAnstgFkt.arrFktAusfg[1]:= stUniAnstgFkt.arrGrdstFkt[1]
										 OR stUniAnstgFkt.arrHandFkt[1]
										 OR stUniAnstgFkt.arrAutomFkt[1];

//****************************************************************************************************
END_ACTION

ACTION b_MittelStellung:
(*Ansteuerungstyp "Mittelstlg." /z.B. Pneumatikzylinder mit ext. Geber...*)

(*Verwendete Softkeytasten = 2 (s.Beispiel)*)

(*       "Handfunktion"       /   "Softkeytaste 1"   /   "Softkeytaste 2"   *)
(*                                                                          *) 
(*------- Stopanschlag -------/______einfahren_______/______ausfahren_______*)

(*Softkeyleiste.1		:Funktion Tastend aktiv /Ventil-0*)
(*Softkeyleiste.2		:Funktion Tastend aktiv /Ventil-1*)

(*Hinweis:
- Funktion wird durch "ResHdBetr" bei Betriebsartenwechsel zurückgenommen
- Funktion wird durch "VerrHdFkt" gesperrt (z.B. bei Kollissionserkennung...)

- Mit "LaufzVorg" kann die Meldelaufzeit angepasst werden (Default: 5sek)
- Mit "VerrMeldg" wird die Meldeausgabe unterdrückt (eventl. Ablaufbedingt)

- Bei "AnstgUntbr" werden die F-Ausgänge deaktiviert (z.B. bei LSG-Unterbr.)
						Erforderlich u.U. bei Sonderbeschaltung einzelner Ausgänge
- Bei "AnstgUng" bleiben die F-Ausgänge auch bei geöffn. Schutzbereich aktiv  
- Bei "AnstgInvt" wird die Logik der Funktions-Ausgänge invertiert  
*)

(**************************************************)	

stUniAnstgFkt.bHandAnw0:= IQ_stUniAnstgHMI.stHandFktHMI[1].bySwitch > 0;
stUniAnstgFkt.bHandAnw1:= IQ_stUniAnstgHMI.stHandFktHMI[2].bySwitch > 0;

IF arrBetrartAutomAktiv[I_nSchutzBer]
	OR I_bResHandFkt
THEN
	stUniAnstgFkt.arrHandFkt[0]:=
	stUniAnstgFkt.arrHandFkt[1]:= FALSE;
ELSE
	IF NOT arrBetrartAutomSpeichn[I_nSchutzBer]
	THEN
		IF NOT arrGrdstlgBetrAktiv[I_nSchutzBer]
		THEN
			IF arrBetrartHandAktiv[I_nSchutzBer]
				AND stUniAnstgFkt.bHandAnw1
				AND NOT I_bVerrHdFkt1
			THEN		
				stUniAnstgFkt.arrHandFkt[1]:= TRUE;
			ELSE
				stUniAnstgFkt.arrHandFkt[1]:= FALSE;	 
			END_IF

			IF arrBetrartHandAktiv[I_nSchutzBer]
				AND stUniAnstgFkt.bHandAnw0
				AND NOT I_bVerrHdFkt0
			THEN		
				stUniAnstgFkt.arrHandFkt[0]:= TRUE;
			ELSE
				stUniAnstgFkt.arrHandFkt[0]:= FALSE;		 
			END_IF
		END_IF
	END_IF
END_IF

(**************************************************)	

IF arrBetrartHandAktiv[I_nSchutzBer]
THEN
	stUniAnstgFkt.arrGrdstFkt[0]:= I_arrZuwGrdstFkt[0];
	stUniAnstgFkt.arrGrdstFkt[1]:= I_arrZuwGrdstFkt[1];
ELSE
	stUniAnstgFkt.arrGrdstFkt[0]:= 
	stUniAnstgFkt.arrGrdstFkt[1]:= FALSE;
END_IF

IF arrBetrartAutomAktiv[I_nSchutzBer] OR TRUE //ToDo
THEN
	stUniAnstgFkt.arrAutomFkt[0]:= I_arrZuwAutomFkt[0];
	stUniAnstgFkt.arrAutomFkt[1]:= I_arrZuwAutomFkt[1];
ELSE
	stUniAnstgFkt.arrAutomFkt[0]:= 
	stUniAnstgFkt.arrAutomFkt[1]:= FALSE;
END_IF

(**************************************************)	

stUniAnstgFkt.arrFktAusfg[0]:= stUniAnstgFkt.arrGrdstFkt[0]
										 OR stUniAnstgFkt.arrHandFkt[0]
										 OR stUniAnstgFkt.arrAutomFkt[0];

stUniAnstgFkt.arrFktAusfg[1]:= stUniAnstgFkt.arrGrdstFkt[1]
										 OR stUniAnstgFkt.arrHandFkt[1]
										 OR stUniAnstgFkt.arrAutomFkt[1];

(**************************************************)
END_ACTION

ACTION c_TestMode:

//****************************************************************************************************
// Zeitintervall für den Testmode erstellen

tReversierZeit	:= TO_TIME(TO_INT(IQ_stUniAnstgHMI.stHandFktHMI[4].sImage));

fbReversierTakt(
	I_bStart	:= bTestModeAktiv,
	I_tBlinkZeit	:= tReversierZeit
);

//****************************************************************************************************
// Handfunktion beschreiben

IF NOT arrBetrartAutomAktiv[I_nSchutzBer]
	AND NOT arrBetrartAutomSpeichn[I_nSchutzBer]
	AND NOT arrGrdstlgBetrAktiv[I_nSchutzBer]
	AND bTestModeAktiv
	AND arrBetrartHandAktiv[I_nSchutzBer]
	AND NOT I_bVerrHdFkt1
	AND NOT I_bVerrHdFkt0
THEN
	IF fbReversierTakt.Q_bOut
	THEN
		stUniAnstgFkt.arrHandFkt[0]:= FALSE;
		stUniAnstgFkt.arrHandFkt[1]:= TRUE;	
	ELSE
		stUniAnstgFkt.arrHandFkt[0]:= TRUE;
		stUniAnstgFkt.arrHandFkt[1]:= FALSE;	
	END_IF
END_IF

//****************************************************************************************************
// Zeitdauer bis erreichen der Endlage messen

rTrigEndlage0(CLK:=I_bZyliAbfrg0);
rTrigEndlage1(CLK:=I_bZyliAbfrg1);

IF rTrigEndlage0.Q
	AND bTestModeAktiv
THEN
	tBisInEndlage0	:= fbReversierTakt.tonBlinker1.ET;
END_IF

IF rTrigEndlage1.Q
	AND bTestModeAktiv
THEN
	tBisInEndlage1	:= fbReversierTakt.tonBlinker2.ET;
END_IF

IF NOT bTestModeAktiv
THEN
	tBisInEndlage1	:= T#0S;
	tBisInEndlage0	:= T#0S;
END_IF

//****************************************************************************************************
// ENDE
END_ACTION

ACTION x_AusgaengeZuweisen:

	(**************************************************)	
	(*Ausgänge zuweisen*)

	CASE I_eAnstgTyp OF
1, 2:	(*Zylindertyp 01: Anstg. 1 Rückstlg. /Abfrg.0*)
		(*Zylindertyp 02: Anstg. 1 Rückstlg. /Abfrg.0-1*)

	Q_bZyliAnstg0:= FALSE;

	Q_bZyliAnstg1:= stUniAnstgFkt.arrFktAusfg[1]
					 	 AND NOT I_bAnstgUntbr
					 	 AND(arrAusgGruppeFrg[I_nSchutzBer]
					 	 OR I_bAnstgUng)
					 	 AND bVersEingAusgAnlagOk;

3, 4:	(*Zylindertyp 03: Anstg. 0-1 Rückstlg. /Abfrg.0*)
		(*Zylindertyp 04: Anstg. 0-1 Rückstlg. /Abfrg.0-1*)

	Q_bZyliAnstg0:= NOT stUniAnstgFkt.arrFktAusfg[1]
					 	 AND NOT I_bAnstgUntbr
					 	 AND(arrAusgGruppeFrg[I_nSchutzBer]
					 	 OR I_bAnstgUng)
					 	 AND bVersEingAusgAnlagOk;

	Q_bZyliAnstg1:= stUniAnstgFkt.arrFktAusfg[1]
					 	 AND NOT I_bAnstgUntbr
					 	 AND(arrAusgGruppeFrg[I_nSchutzBer]
					 	 OR I_bAnstgUng)
					 	 AND bVersEingAusgAnlagOk;

5, 6:	(*Zylindertyp 05: Anstg. 0-1 Impulsstlg. /Abfrg.0*)
		(*Zylindertyp 06: Anstg. 0-1 Impulsstlg. /Abfrg.0-1*)

	Q_bZyliAnstg0:= NOT stUniAnstgFkt.arrFktAusfg[1]
					 	 AND NOT I_bAnstgUntbr
					 	 AND NOT I_bZyliAbfrg0
					 	 AND (arrAusgGruppeFrg[I_nSchutzBer]
				    	 OR I_bAnstgUng)
					 	 AND bVersEingAusgAnlagOk;

	Q_bZyliAnstg1:= stUniAnstgFkt.arrFktAusfg[1]
					 	 AND NOT I_bAnstgUntbr
					 	 AND NOT I_bZyliAbfrg1
					 	 AND (arrAusgGruppeFrg[I_nSchutzBer]
				    	 OR I_bAnstgUng)
					 	 AND bVersEingAusgAnlagOk;

7:		(*Zylindertyp 07: Anstg. 0-1 Mittelstlg. /Abfrg.0-1*)

	Q_bZyliAnstg0:= stUniAnstgFkt.arrFktAusfg[0]
					 	 AND NOT I_bAnstgUntbr
					 	 AND (arrAusgGruppeFrg[I_nSchutzBer]
				    	 OR I_bAnstgUng)
					 	 AND bVersEingAusgAnlagOk;

	Q_bZyliAnstg1:= stUniAnstgFkt.arrFktAusfg[1]
					 	 AND NOT I_bAnstgUntbr
					 	 AND (arrAusgGruppeFrg[I_nSchutzBer]
				    	 OR I_bAnstgUng)
					 	 AND bVersEingAusgAnlagOk;
	END_CASE

	(**************************************************)	
	(*Ausgänge invertieren*)

	IF I_bAnstgInvt THEN
		Q_bZyliAnstg0:= NOT Q_bZyliAnstg0;
		Q_bZyliAnstg1:= NOT Q_bZyliAnstg1;
	END_IF

	(**************************************************)
END_ACTION

ACTION y_ZustaendeAnzeigen:
	
//****************************************************************************************************
// Zustände anzeigen

CASE I_eAnstgDef OF

eZyliDef0Def1, eZyliDef1Def0:
	sTextHandFkt1[0]:= I_sZuDef0;
	sTextHandFkt1[1]:= I_sInDef0;
	sTextHandFkt2[0]:= I_sZuDef1;
	sTextHandFkt2[1]:= I_sInDef1;
eZyliGrdArbstlg,eZyliArbGrdstlg:
	sTextHandFkt1[0]:= 'zur Grundstlg.';
	sTextHandFkt1[1]:= 'in Grundstlg.';
	sTextHandFkt2[0]:= 'zur Arbeitstlg.';
	sTextHandFkt2[1]:= 'in Arbeitstlg.';
eZyliAbsAnheb,eZyliAnhAbsenk:
	sTextHandFkt1[0]:= 'absenken';
	sTextHandFkt1[1]:= 'abgesenkt';
	sTextHandFkt2[0]:= 'anheben';
	sTextHandFkt2[1]:= 'angehoben';
eZyliEinAusfahr,eZyliAusEinfahr:
	sTextHandFkt1[0]:= 'einfahren';
	sTextHandFkt1[1]:= 'eingefahren';
	sTextHandFkt2[0]:= 'ausfahren';
	sTextHandFkt2[1]:= 'ausgefahren';
eZyliZurVorfahr,eZyliVorZurfahr:
	sTextHandFkt1[0]:= 'zurückfahren';
	sTextHandFkt1[1]:= 'zurückgefahren';
	sTextHandFkt2[0]:= 'vorfahren';
	sTextHandFkt2[1]:= 'vorgefahren';
eZyliEinAussteun,eZyliAusEinsteun:
	sTextHandFkt1[0]:= 'einsteuern';
	sTextHandFkt1[1]:= 'eingesteuert';
	sTextHandFkt2[0]:= 'aussteuern';
	sTextHandFkt2[1]:= 'ausgesteuert';
eZyliLoesSpann,eZyliSpannLoes:
	sTextHandFkt1[0]:= 'lösen';
	sTextHandFkt1[1]:= 'gelöst';
	sTextHandFkt2[0]:= 'spannen';
	sTextHandFkt2[1]:= 'gespannt';
eZyliOeffnSchliess,eZyliSchliessOeffn:
	sTextHandFkt1[0]:= 'öffnen';
	sTextHandFkt1[1]:= 'geöffnet';
	sTextHandFkt2[0]:= 'schliessen';
	sTextHandFkt2[1]:= 'geschlossen';
eZyliZu0Zu180,eZyliZu180Zu0:
	sTextHandFkt1[0]:= 'zu 0°';
	sTextHandFkt1[1]:= 'in 0°';
	sTextHandFkt2[0]:= 'zu 180°';
	sTextHandFkt2[1]:= 'in 180°';
END_CASE
	
//****************************************************************************************************
// Tasten beschriften und Zustand und Farben ändern

IF I_eAnstgDef >= 50 //Zuweisungen tauschen 
THEN
	sTextHandFktX:= sTextHandFkt1; 
	sTextHandFkt1:= sTextHandFkt2;
	sTextHandFkt2:= sTextHandFktX;
END_IF

IF NOT stUniAnstgFkt.arrHandFkt[1]
THEN	// Handfunktion.1 aktiv
	IF Q_bZyliAnstg0
		AND NOT I_bZyliAbfrg0
	THEN	// Zylinder nach links "unterwegs"
		IQ_stUniAnstgHMI.stHandFktHMI[1].sColour:= cGelbAsString;
		IQ_stUniAnstgHMI.stHandFktHMI[1].iDisplayMode:= 1;
		IQ_stUniAnstgHMI.stHandFktHMI[1].sText:= sTextHandFkt1[0];
	ELSE	// Zylinder in Position links angekommen
		IQ_stUniAnstgHMI.stHandFktHMI[1].sColour:= cGruenAsString;
		IQ_stUniAnstgHMI.stHandFktHMI[1].iDisplayMode:= 0;
		IQ_stUniAnstgHMI.stHandFktHMI[1].sText:= sTextHandFkt1[1];
	END_IF
ELSE	// Handfunktion links nicht aktiv
	IQ_stUniAnstgHMI.stHandFktHMI[1].sColour		:= cDefaultAsString;
	IQ_stUniAnstgHMI.stHandFktHMI[1].sText			:= sTextHandFkt1[0];
	IQ_stUniAnstgHMI.stHandFktHMI[1].iDisplayMode:= 1;
END_IF

IF stUniAnstgFkt.arrHandFkt[1]
THEN	// Handfunktion.2 aktiv
	IF Q_bZyliAnstg1
		AND NOT I_bZyliAbfrg1
	THEN	// Zylinder nach rechts "unterwegs"
		IQ_stUniAnstgHMI.stHandFktHMI[2].sColour:= cGelbAsString;
		IQ_stUniAnstgHMI.stHandFktHMI[2].iDisplayMode:= 1;
		IQ_stUniAnstgHMI.stHandFktHMI[2].sText:= sTextHandFkt2[0];
	ELSE	// Zylinder in Position rechts angekommen
		IQ_stUniAnstgHMI.stHandFktHMI[2].sColour:= cGruenAsString;
		IQ_stUniAnstgHMI.stHandFktHMI[2].iDisplayMode:= 0;
		IQ_stUniAnstgHMI.stHandFktHMI[2].sText:= sTextHandFkt2[1];
	END_IF
ELSE	// Handfunktion rechts nicht aktiv
	IQ_stUniAnstgHMI.stHandFktHMI[2].sColour		:= cDefaultAsString;
	IQ_stUniAnstgHMI.stHandFktHMI[2].sText			:= sTextHandFkt2[0];
	IQ_stUniAnstgHMI.stHandFktHMI[2].iDisplayMode:= 1;
END_IF

// Testmode umschalten
rTrigTestMode(CLK:= IQ_stUniAnstgHMI.stHandFktHMI[3].bySwitch > 0);

IF rTrigTestMode.Q
THEN
	bTestModeAktiv	:= NOT bTestModeAktiv;
END_IF

IF NOT arrBetrartHandAktiv[I_nSchutzBer]
	OR IQ_stUniAnstgHMI.stHandFktHMI[1].bySwitch > 0
	OR IQ_stUniAnstgHMI.stHandFktHMI[2].bySwitch > 0
THEN	// Wenn eine Handfunktionstaste aktiviert wird, dann geht der Testmode aus.
	bTestModeAktiv	:= FALSE;
END_IF

IF bTestModeAktiv
THEN
	IQ_stUniAnstgHMI.stHandFktHMI[5].sText	:= CONCAT('Zeit bis Endlage0: ',TO_STRING(tBisInEndlage0));
	IQ_stUniAnstgHMI.stHandFktHMI[6].sText	:= CONCAT('Zeit bis Endlage1: ',TO_STRING(tBisInEndlage1));
ELSE
	IQ_stUniAnstgHMI.stHandFktHMI[5].sText	:= '';	// Wenn die Taste nicht beschriebn ist, wird sie ausgeblendet
	IQ_stUniAnstgHMI.stHandFktHMI[6].sText	:= '';	// Wenn die Taste nicht beschriebn ist, wird sie ausgeblendet
END_IF

IF bTestModeAktiv
THEN
	IQ_stUniAnstgHMI.stHandFktHMI[3].sColour	:= cBlauAsString;
	IQ_stUniAnstgHMI.stHandFktHMI[3].iDisplayMode:= 1;
ELSE
	IQ_stUniAnstgHMI.stHandFktHMI[3].sColour	:= cDefaultAsString;
	IQ_stUniAnstgHMI.stHandFktHMI[3].iDisplayMode:= 0;
END_IF

IF NOT bTestModeZylinder
THEN
	bTestModeAktiv := FALSE;
	IQ_stUniAnstgHMI.stHandFktHMI[3].sText	:= '';
	IQ_stUniAnstgHMI.stHandFktHMI[4].sText	:= '';
	IQ_stUniAnstgHMI.stHandFktHMI[5].sText	:= '';
	IQ_stUniAnstgHMI.stHandFktHMI[6].sText	:= '';
ELSE
	IQ_stUniAnstgHMI.stHandFktHMI[4].sText	:= 'Zeit in ms';
	IQ_stUniAnstgHMI.stHandFktHMI[3].sText	:= 'Testmode';
END_IF

IQ_stUniAnstgHMI.stHandFktHMI[4].byStatus	:= 0;	// Muss immer beschreibbar sein
IQ_stUniAnstgHMI.stHandFktHMI[5].sColour	:= cDefaultAsString;
IQ_stUniAnstgHMI.stHandFktHMI[6].sColour	:= cDefaultAsString;
IQ_stUniAnstgHMI.stHandFktHMI[5].byStatus	:= 1;	// Diese Tasten sind immer gesperrt. Ist nur eine Anzeige
IQ_stUniAnstgHMI.stHandFktHMI[6].byStatus	:= 1;	// Diese Tasten sind immer gesperrt. Ist nur eine Anzeige

//****************************************************************************************************
// Tastenzustand
IF NOT arrBetrartHandAktiv[I_nSchutzBer]
THEN	// Funktionen sperren
	IQ_stUniAnstgHMI.stHandFktHMI[1].byStatus	:=
	IQ_stUniAnstgHMI.stHandFktHMI[2].byStatus	:=
	IQ_stUniAnstgHMI.stHandFktHMI[3].byStatus	:= 1;	// Testmode sperren
	IQ_stUniAnstgHMI.stHandFktHMI[1].sText	:= sTextHandFkt1[0];
	IQ_stUniAnstgHMI.stHandFktHMI[2].sText	:= sTextHandFkt2[0];
ELSE	// Funktionen freigeben
	IQ_stUniAnstgHMI.stHandFktHMI[1].byStatus.0	:= I_bVerrHdFkt0;
	IQ_stUniAnstgHMI.stHandFktHMI[2].byStatus.0	:= I_bVerrHdFkt1;
	IQ_stUniAnstgHMI.stHandFktHMI[3].byStatus.0	:= FALSE;	// Testmode freigeben
END_IF

//****************************************************************************************************
END_ACTION

ACTION z_FehlerMeldung:
	
//****************************************************************************************************
// Meldungen ausgeben

	CASE I_eAnstgTyp OF
1:		(*Zylindertyp 01: Anstg. 1 Rückstlg. /Abfrg.0*)

	fbLfzMeldAusg.I_bLaufzAnstg0:=	NOT Q_bZyliAnstg1;
	fbLfzMeldAusg.I_bLaufzAbfrg0:=	I_bZyliAbfrg0;
	fbLfzMeldAusg.I_bLaufzAnstg1:=	Q_bZyliAnstg1;
	fbLfzMeldAusg.I_bLaufzAbfrg1:=	NOT I_bZyliAbfrg0;

2:		(*Zylindertyp 02: Anstg. 1 Rückstlg. /Abfrg.0-1*)

	fbLfzMeldAusg.I_bLaufzAnstg0:=	NOT Q_bZyliAnstg1;
	fbLfzMeldAusg.I_bLaufzAbfrg0:=	I_bZyliAbfrg0;
	fbLfzMeldAusg.I_bLaufzAnstg1:=	Q_bZyliAnstg1;
	fbLfzMeldAusg.I_bLaufzAbfrg1:=	I_bZyliAbfrg1;

3, 5:	(*Zylindertyp 03: Anstg. 0-1 Rückstlg. /Abfrg.0*)
		(*Zylindertyp 05: Anstg. 0-1 Impulsstlg. /Abfrg.0*)

	fbLfzMeldAusg.I_bLaufzAnstg0:=	Q_bZyliAnstg0;
	fbLfzMeldAusg.I_bLaufzAbfrg0:=	I_bZyliAbfrg0;
	fbLfzMeldAusg.I_bLaufzAnstg1:=	Q_bZyliAnstg1;
	fbLfzMeldAusg.I_bLaufzAbfrg1:=	NOT I_bZyliAbfrg0;

4, 6:	(*Zylindertyp 04: Anstg. 0-1 Rückstlg. /Abfrg.0-1*)
		(*Zylindertyp 06: Anstg. 0-1 Impulsstlg. /Abfrg.0-1*)

	fbLfzMeldAusg.I_bLaufzAnstg0:=	Q_bZyliAnstg0;
	fbLfzMeldAusg.I_bLaufzAbfrg0:=	I_bZyliAbfrg0;
	fbLfzMeldAusg.I_bLaufzAnstg1:=	Q_bZyliAnstg1;
	fbLfzMeldAusg.I_bLaufzAbfrg1:=	I_bZyliAbfrg1;

7:		(*Zylindertyp 07: Anstg. 0-1 Mittelstlg. /Abfrg.0-1*)
	
	fbLfzMeldAusg.I_bLaufzAnstg0:=	Q_bZyliAnstg0;
	fbLfzMeldAusg.I_bLaufzAbfrg0:=	I_bZyliAbfrg0;
	fbLfzMeldAusg.I_bLaufzAnstg1:=	Q_bZyliAnstg1;
	fbLfzMeldAusg.I_bLaufzAbfrg1:=	I_bZyliAbfrg1;
	END_CASE

	fbLfzMeldAusg (I_bMeldgFreig	:= arrAusgGruppeFrg[I_nSchutzBer]
								   			AND bVersEingAusgAnlagOk
								   			AND NOT I_bVerrMeldg,
				  	   I_tLaufzDauer	:= I_tLaufzVorg);	(*Defaultwert = 5sek*)
		
	IQ_stUniAnstgHMI.stMeldAusgHMI.SourceID			:= 0;	// Nicht mehr verwendet
	IQ_stUniAnstgHMI.stMeldAusgHMI.SourceName			:= I_sStatName;
	IQ_stUniAnstgHMI.stMeldAusgHMI.sAktorName			:= I_sAktorName;
	IF I_eAnstgDef >= 20 //Zuweisungen tauschen 
		THEN
			IF I_sAktorBMK1 <> ''
			THEN	// I_sAktorBMK ist beschrieben. Damit wird der String als BMK genommen
 				IQ_stUniAnstgHMI.stMeldAusgHMI.sBMK0	:= I_sAktorBMK1;
			ELSE	// Der Kommentar von VARINFO wird als BMK genommen
				IQ_stUniAnstgHMI.stMeldAusgHMI.sBMK0	:= I_stVarInfoBMK1.Comment;
			END_IF
			IF I_sAktorBMK0 <> ''
			THEN	// I_sAktorBMK ist beschrieben. Damit wird der String als BMK genommen
 				IQ_stUniAnstgHMI.stMeldAusgHMI.sBMK1	:= I_sAktorBMK0;
			ELSE	// Der Kommentar von VARINFO wird als BMK genommen
				IQ_stUniAnstgHMI.stMeldAusgHMI.sBMK1	:= I_stVarInfoBMK0.Comment;
			END_IF

			bLaufzMeldg0:= fbLfzMeldAusg.Q_bLaufzMeldg1 AND NOT I_bVerrMeldg1;
			bLaufzMeldg1:= fbLfzMeldAusg.Q_bLaufzMeldg0 AND NOT I_bVerrMeldg0;
		ELSE
			IF I_sAktorBMK0 <> ''
			THEN	// I_sAktorBMK ist beschrieben. Damit wird der String als BMK genommen
 				IQ_stUniAnstgHMI.stMeldAusgHMI.sBMK1	:= I_sAktorBMK1;
			ELSE	// Der Kommentar von VARINFO wird als BMK genommen
				IQ_stUniAnstgHMI.stMeldAusgHMI.sBMK1	:= I_stVarInfoBMK1.Comment;
			END_IF
			IF I_sAktorBMK1 <> ''
			THEN	// I_sAktorBMK ist beschrieben. Damit wird der String als BMK genommen
 				IQ_stUniAnstgHMI.stMeldAusgHMI.sBMK0	:= I_sAktorBMK0;
			ELSE	// Der Kommentar von VARINFO wird als BMK genommen
				IQ_stUniAnstgHMI.stMeldAusgHMI.sBMK0	:= I_stVarInfoBMK0.Comment;
			END_IF
			bLaufzMeldg0:= fbLfzMeldAusg.Q_bLaufzMeldg0 AND NOT I_bVerrMeldg0;
			bLaufzMeldg1:= fbLfzMeldAusg.Q_bLaufzMeldg1 AND NOT I_bVerrMeldg1;
	END_IF
	
	CASE I_eAnstgDef OF
eZyliDef0Def1, eZyliDef1Def0:
	IQ_stUniAnstgHMI.stMeldAusgHMI.bLfzMeldAusgDef0	:= bLaufzMeldg0
																		OR bTestMeldZyl;
	IQ_stUniAnstgHMI.stMeldAusgHMI.bLfzMeldAusgDef1	:= bLaufzMeldg1
																		OR bTestMeldZyl; 
	IQ_stUniAnstgHMI.stMeldAusgHMI.bMeldSensFehlDef	:= fbLfzMeldAusg.Q_bSensMeldg
																		OR bTestMeldZyl;
	IQ_stUniAnstgHMI.stMeldAusgHMI.sLzFehlerDef0		:= I_sLzFehlerDef0;
	IQ_stUniAnstgHMI.stMeldAusgHMI.sLzFehlerDef1		:= I_sLzFehlerDef1; 
	IQ_stUniAnstgHMI.stMeldAusgHMI.sSensorFehlDef	:= I_sSensorFehlDef;
eZyliGrdArbstlg,eZyliArbGrdstlg:
	IQ_stUniAnstgHMI.stMeldAusgHMI.bLfzMeldAusg01	:= bLaufzMeldg0
																		OR bTestMeldZyl;
	IQ_stUniAnstgHMI.stMeldAusgHMI.bLfzMeldAusg11	:= bLaufzMeldg1
																		OR bTestMeldZyl; 
	IQ_stUniAnstgHMI.stMeldAusgHMI.bMeldSensFehl1	:= fbLfzMeldAusg.Q_bSensMeldg
																		OR bTestMeldZyl; 
eZyliAbsAnheb,eZyliAnhAbsenk:
	IQ_stUniAnstgHMI.stMeldAusgHMI.bLfzMeldAusg02	:= bLaufzMeldg0
																		OR bTestMeldZyl;
	IQ_stUniAnstgHMI.stMeldAusgHMI.bLfzMeldAusg12	:= bLaufzMeldg1
																		OR bTestMeldZyl; 
	IQ_stUniAnstgHMI.stMeldAusgHMI.bMeldSensFehl2	:= fbLfzMeldAusg.Q_bSensMeldg
																		OR bTestMeldZyl; 
eZyliEinAusfahr,eZyliAusEinfahr:
	IQ_stUniAnstgHMI.stMeldAusgHMI.bLfzMeldAusg03	:= bLaufzMeldg0
																		OR bTestMeldZyl;
	IQ_stUniAnstgHMI.stMeldAusgHMI.bLfzMeldAusg13	:= bLaufzMeldg1
																		OR bTestMeldZyl; 
	IQ_stUniAnstgHMI.stMeldAusgHMI.bMeldSensFehl3	:= fbLfzMeldAusg.Q_bSensMeldg
																		OR bTestMeldZyl; 
eZyliZurVorfahr,eZyliVorZurfahr:
	IQ_stUniAnstgHMI.stMeldAusgHMI.bLfzMeldAusg04	:= bLaufzMeldg0
																		OR bTestMeldZyl;
	IQ_stUniAnstgHMI.stMeldAusgHMI.bLfzMeldAusg14	:= bLaufzMeldg1
																		OR bTestMeldZyl; 
	IQ_stUniAnstgHMI.stMeldAusgHMI.bMeldSensFehl4	:= fbLfzMeldAusg.Q_bSensMeldg
																		OR bTestMeldZyl; 
eZyliEinAussteun,eZyliAusEinsteun:
	IQ_stUniAnstgHMI.stMeldAusgHMI.bLfzMeldAusg05	:= bLaufzMeldg0
																		OR bTestMeldZyl;
	IQ_stUniAnstgHMI.stMeldAusgHMI.bLfzMeldAusg15	:= bLaufzMeldg1
																		OR bTestMeldZyl; 
	IQ_stUniAnstgHMI.stMeldAusgHMI.bMeldSensFehl5	:= fbLfzMeldAusg.Q_bSensMeldg
																		OR bTestMeldZyl; 
eZyliLoesSpann,eZyliSpannLoes:
	IQ_stUniAnstgHMI.stMeldAusgHMI.bLfzMeldAusg06	:= bLaufzMeldg0
																		OR bTestMeldZyl;
	IQ_stUniAnstgHMI.stMeldAusgHMI.bLfzMeldAusg16	:= bLaufzMeldg1
																		OR bTestMeldZyl; 
	IQ_stUniAnstgHMI.stMeldAusgHMI.bMeldSensFehl6	:= fbLfzMeldAusg.Q_bSensMeldg
																		OR bTestMeldZyl; 
eZyliOeffnSchliess,eZyliSchliessOeffn:
	IQ_stUniAnstgHMI.stMeldAusgHMI.bLfzMeldAusg07	:= bLaufzMeldg0
																		OR bTestMeldZyl;
	IQ_stUniAnstgHMI.stMeldAusgHMI.bLfzMeldAusg17	:= bLaufzMeldg1
																		OR bTestMeldZyl; 
	IQ_stUniAnstgHMI.stMeldAusgHMI.bMeldSensFehl7	:= fbLfzMeldAusg.Q_bSensMeldg
																		OR bTestMeldZyl;
eZyliZu0Zu180,eZyliZu180Zu0:
	IQ_stUniAnstgHMI.stMeldAusgHMI.bLfzMeldAusg09	:= bLaufzMeldg0
																		OR bTestMeldZyl;
	IQ_stUniAnstgHMI.stMeldAusgHMI.bLfzMeldAusg19	:= bLaufzMeldg1
																		OR bTestMeldZyl; 
	IQ_stUniAnstgHMI.stMeldAusgHMI.bMeldSensFehl9	:= fbLfzMeldAusg.Q_bSensMeldg
																		OR bTestMeldZyl;
	END_CASE
	
	IQ_stUniAnstgHMI.stMeldAusgHMI.bMeldHinweis		:= FALSE;	

	IF fbLfzMeldAusg.Q_bSensMeldg THEN
		bSensFehlAllgVorhand:= TRUE;
	END_IF

//****************************************************************************************************
END_ACTION

END_FUNCTION_BLOCK
